C07295=1221.283,24.930,-43.229,-179.294,5.443,148.738
C07296=1221.289,24.681,-43.214,-179.297,5.442,148.739
C07297=1221.293,24.432,-43.199,-179.299,5.442,148.739
C07298=1221.299,24.182,-43.183,-179.302,5.441,148.740
C07299=1221.303,23.932,-43.168,-179.304,5.442,148.741
C07300=1221.308,23.682,-43.153,-179.307,5.441,148.741
C07301=1221.314,23.433,-43.137,-179.309,5.441,148.742
C07302=1221.318,23.184,-43.122,-179.312,5.440,148.743
C07303=1221.324,22.934,-43.107,-179.315,5.439,148.743
C07304=1221.328,22.685,-43.091,-179.317,5.439,148.744
C07305=1221.333,22.435,-43.076,-179.320,5.438,148.745
C07306=1221.338,22.186,-43.061,-179.321,5.438,148.745
C07307=1221.343,21.936,-43.046,-179.324,5.438,148.746
C07308=1221.348,21.687,-43.031,-179.327,5.437,148.747
C07309=1221.354,21.438,-43.015,-179.329,5.437,148.747
C07310=1221.358,21.188,-43.000,-179.332,5.436,148.748
C07311=1221.363,20.938,-42.985,-179.335,5.436,148.749
C07312=1221.368,20.689,-42.970,-179.337,5.436,148.749
C07313=1221.373,20.439,-42.955,-179.339,5.435,148.750
C07314=1221.378,20.190,-42.940,-179.342,5.435,148.751
C07315=1221.384,19.940,-42.925,-179.345,5.434,148.751
C07316=1221.388,19.691,-42.910,-179.347,5.434,148.752
C07317=1221.393,19.441,-42.894,-179.350,5.433,148.753
C07318=1221.398,19.192,-42.879,-179.353,5.433,148.753
C07319=1221.403,18.942,-42.864,-179.354,5.433,148.754
C07320=1221.408,18.693,-42.849,-179.357,5.432,148.755
C07321=1221.413,18.443,-42.833,-179.359,5.432,148.755
C07322=1221.418,18.194,-42.819,-179.362,5.431,148.756
C07323=1221.423,17.945,-42.804,-179.365,5.431,148.757
C07324=1221.428,17.695,-42.788,-179.367,5.430,148.757
C07325=1221.433,17.446,-42.774,-179.370,5.430,148.758
C07326=1221.439,17.196,-42.759,-179.372,5.430,148.759
C07327=1221.443,16.946,-42.743,-179.375,5.429,148.759
C07328=1221.449,16.696,-42.728,-179.377,5.429,148.760
C07329=1221.453,16.447,-42.713,-179.380,5.428,148.761
C07330=1221.458,16.198,-42.698,-179.383,5.428,148.761
C07331=1221.464,15.948,-42.683,-179.385,5.428,148.762
C07332=1221.468,15.699,-42.668,-179.387,5.427,148.763
C07333=1221.473,15.449,-42.654,-179.390,5.426,148.763
C07334=1221.479,15.200,-42.639,-179.392,5.426,148.764
C07335=1221.483,14.951,-42.624,-179.395,5.425,148.765
C07336=1221.489,14.701,-42.609,-179.397,5.426,148.765
C07337=1221.493,14.452,-42.594,-179.400,5.425,148.766
C07338=1221.498,14.202,-42.579,-179.402,5.425,148.767
C07339=1221.504,13.953,-42.564,-179.405,5.424,148.767
C07340=1221.509,13.703,-42.550,-179.408,5.424,148.768
C07341=1221.513,13.454,-42.535,-179.410,5.423,148.769
C07342=1221.519,13.204,-42.519,-179.412,5.423,148.769
C07343=1221.523,12.954,-42.504,-179.415,5.423,148.770
C07344=1221.528,12.705,-42.489,-179.418,5.422,148.771
C07345=1221.534,12.455,-42.474,-179.420,5.422,148.771
C07346=1221.538,12.206,-42.459,-179.423,5.421,148.772
C07347=1221.543,11.956,-42.445,-179.425,5.421,148.773
C07348=1221.548,11.707,-42.430,-179.428,5.421,148.773
C07349=1221.553,11.457,-42.415,-179.430,5.420,148.774
C07350=1221.558,11.207,-42.401,-179.432,5.420,148.775
C07351=1221.563,10.958,-42.386,-179.435,5.419,148.775
C07352=1221.569,10.708,-42.371,-179.437,5.419,148.776
C07353=1221.573,10.459,-42.356,-179.440,5.419,148.777
C07354=1221.578,10.209,-42.342,-179.442,5.418,148.777
C07355=1221.583,9.960,-42.327,-179.445,5.418,148.778
C07356=1221.589,9.710,-42.312,-179.448,5.417,148.779
C07357=1221.593,9.461,-42.297,-179.450,5.417,148.779
C07358=1221.598,9.211,-42.283,-179.452,5.417,148.780
C07359=1221.604,8.962,-42.269,-179.455,5.416,148.781
C07360=1221.609,8.713,-42.253,-179.458,5.416,148.781
C07361=1221.614,8.463,-42.239,-179.460,5.415,148.782
C07362=1221.619,8.214,-42.225,-179.463,5.416,148.783
C07363=1221.624,7.964,-42.210,-179.465,5.415,148.784
C07364=1221.629,7.715,-42.195,-179.468,5.415,148.784
C07365=1221.634,7.465,-42.180,-179.470,5.414,148.785
C07366=1221.639,7.216,-42.166,-179.473,5.414,148.786
C07367=1221.644,6.966,-42.151,-179.475,5.414,148.786
C07368=1221.649,6.717,-42.136,-179.477,5.413,148.787
C07369=1221.654,6.467,-42.122,-179.480,5.412,148.787
C07370=1221.659,6.217,-42.108,-179.483,5.412,148.788
C07371=1221.664,5.967,-42.093,-179.485,5.411,148.789
C07372=1221.669,5.718,-42.078,-179.487,5.412,148.789
C07373=1221.674,5.469,-42.064,-179.490,5.411,148.790
C07374=1221.679,5.219,-42.049,-179.493,5.411,148.791
C07375=1221.684,4.970,-42.034,-179.495,5.410,148.792
C07376=1221.689,4.721,-42.020,-179.497,5.410,148.792
C07377=1221.695,4.471,-42.006,-179.500,5.410,148.793
C07378=1221.700,4.221,-41.991,-179.503,5.409,148.794
C07379=1221.704,3.972,-41.976,-179.505,5.409,148.794
C07380=1221.710,3.703,-41.961,-179.508,5.408,148.795
C07381=1221.715,3.434,-41.946,-179.511,5.408,148.796
C07382=1221.720,3.165,-41.930,-179.514,5.408,148.797
C07383=1221.726,2.895,-41.914,-179.516,5.408,148.797
C07384=1221.731,2.646,-41.899,-179.519,5.407,148.798
C07385=1221.736,2.396,-41.885,-179.521,5.407,148.799
C07386=1221.741,2.147,-41.871,-179.524,5.406,148.799
C07387=1221.746,1.898,-41.857,-179.527,5.406,148.800
C07388=1221.751,1.648,-41.843,-179.529,5.406,148.801
C07389=1221.756,1.399,-41.828,-179.531,5.405,148.801
C07390=1221.761,1.149,-41.813,-179.533,5.405,148.802
C07391=1221.766,0.900,-41.799,-179.536,5.404,148.803
C07392=1221.771,0.650,-41.785,-179.538,5.405,148.803
C07393=1221.776,0.401,-41.771,-179.541,5.404,148.804
C07394=1221.781,0.151,-41.757,-179.543,5.404,148.805
C07395=1221.786,-0.099,-41.742,-179.546,5.403,148.805
C07396=1221.791,-0.348,-41.728,-179.548,5.403,148.806
C07397=1221.796,-0.597,-41.713,-179.551,5.403,148.807
C07398=1221.801,-0.847,-41.699,-179.553,5.402,148.807
C07399=1221.806,-1.096,-41.685,-179.556,5.402,148.808
C07400=1221.811,-1.346,-41.671,-179.558,5.402,148.809
C07401=1221.816,-1.596,-41.656,-179.561,5.402,148.809
C07402=1221.821,-1.845,-41.642,-179.563,5.401,148.810
C07403=1221.826,-2.095,-41.628,-179.566,5.400,148.811
C07404=1221.832,-2.344,-41.614,-179.568,5.401,148.811
C07405=1221.837,-2.594,-41.600,-179.571,5.400,148.812
C07406=1221.842,-2.843,-41.585,-179.574,5.400,148.813
C07407=1221.847,-3.093,-41.571,-179.576,5.399,148.814
C07408=1221.852,-3.343,-41.557,-179.578,5.400,148.814
C07409=1221.857,-3.592,-41.543,-179.581,5.399,148.815
C07410=1221.862,-3.842,-41.529,-179.584,5.399,148.816
C07411=1221.867,-4.091,-41.514,-179.586,5.398,148.816
C07412=1221.872,-4.341,-41.500,-179.588,5.398,148.817
C07413=1221.877,-4.591,-41.486,-179.591,5.398,148.818
C07414=1221.883,-4.840,-41.472,-179.594,5.397,148.818
C07415=1221.887,-5.089,-41.458,-179.596,5.397,148.819
C07416=1221.892,-5.339,-41.443,-179.598,5.397,148.820
C07417=1221.897,-5.589,-41.429,-179.601,5.396,148.820
C07418=1221.902,-5.838,-41.416,-179.603,5.396,148.821
C07419=1221.907,-6.087,-41.401,-179.606,5.395,148.822
C07420=1221.912,-6.337,-41.387,-179.608,5.395,148.822
C07421=1221.917,-6.587,-41.374,-179.611,5.395,148.823
C07422=1221.923,-6.836,-41.360,-179.613,5.394,148.824
C07423=1221.928,-7.086,-41.345,-179.616,5.394,148.824
C07424=1221.933,-7.336,-41.331,-179.618,5.394,148.825
C07425=1221.938,-7.585,-41.317,-179.621,5.394,148.826
C07426=1221.943,-7.834,-41.303,-179.623,5.393,148.826
C07427=1221.948,-8.084,-41.289,-179.626,5.393,148.827
C07428=1221.953,-8.334,-41.275,-179.628,5.393,148.828
C07429=1221.958,-8.583,-41.261,-179.631,5.392,148.829
C07430=1221.963,-8.833,-41.247,-179.633,5.392,148.829
C07431=1221.968,-9.083,-41.233,-179.635,5.392,148.830
C07432=1221.973,-9.332,-41.219,-179.638,5.392,148.831
C07433=1221.978,-9.581,-41.206,-179.641,5.391,148.831
C07434=1221.983,-9.831,-41.191,-179.643,5.391,148.832
C07435=1221.988,-10.081,-41.178,-179.645,5.391,148.833
C07436=1221.994,-10.330,-41.164,-179.648,5.391,148.833
C07437=1221.999,-10.580,-41.150,-179.651,5.390,148.834
C07438=1222.003,-10.829,-41.136,-179.653,5.390,148.835
C07439=1222.008,-11.079,-41.122,-179.655,5.390,148.835
C07440=1222.014,-11.328,-41.108,-179.658,5.389,148.836
C07441=1222.019,-11.578,-41.094,-179.661,5.389,148.837
C07442=1222.023,-11.828,-41.080,-179.663,5.389,148.838
C07443=1222.029,-12.077,-41.067,-179.666,5.389,148.838
C07444=1222.034,-12.327,-41.053,-179.668,5.388,148.839
C07445=1222.039,-12.577,-41.039,-179.671,5.388,148.840
C07446=1222.044,-12.825,-41.025,-179.673,5.388,148.840
C07447=1222.049,-13.076,-41.012,-179.676,5.387,148.841
C07448=1222.054,-13.325,-40.998,-179.678,5.387,148.842
C07449=1222.059,-13.574,-40.984,-179.680,5.387,148.842
C07450=1222.064,-13.824,-40.970,-179.683,5.387,148.843
C07451=1222.069,-14.073,-40.957,-179.686,5.386,148.844
C07452=1222.074,-14.323,-40.942,-179.688,5.386,148.844
C07453=1222.079,-14.573,-40.928,-179.690,5.386,148.845
C07454=1222.084,-14.822,-40.916,-179.693,5.385,148.846
C07455=1222.089,-15.072,-40.901,-179.696,5.385,148.847
C07456=1222.094,-15.322,-40.887,-179.698,5.385,148.847
C07457=1222.099,-15.571,-40.874,-179.700,5.384,148.848
C07458=1222.104,-15.821,-40.860,-179.703,5.384,148.848
C07459=1222.110,-16.070,-40.847,-179.705,5.384,148.849
C07460=1222.115,-16.320,-40.833,-179.707,5.384,148.850
C07461=1222.119,-16.569,-40.819,-179.710,5.383,148.850
C07462=1222.125,-16.819,-40.806,-179.713,5.383,148.851
C07463=1222.130,-17.068,-40.792,-179.715,5.383,148.852
C07464=1222.135,-17.318,-40.779,-179.717,5.383,148.853
C07465=1222.140,-17.568,-40.765,-179.720,5.382,148.853
C07466=1222.145,-17.817,-40.751,-179.722,5.382,148.854
C07467=1222.150,-18.067,-40.738,-179.725,5.382,148.855
C07468=1222.155,-18.316,-40.723,-179.727,5.381,148.855
C07469=1222.161,-18.566,-40.711,-179.729,5.382,148.856
C07470=1222.165,-18.815,-40.697,-179.732,5.381,148.857
C07471=1222.171,-19.065,-40.683,-179.735,5.381,148.857
C07472=1222.176,-19.315,-40.670,-179.737,5.380,148.858
C07473=1222.181,-19.565,-40.656,-179.740,5.380,148.859
C07474=1222.186,-19.814,-40.643,-179.742,5.380,148.860
C07475=1222.191,-20.064,-40.629,-179.745,5.379,148.860
C07476=1222.196,-20.313,-40.615,-179.747,5.380,148.861
C07477=1222.201,-20.563,-40.602,-179.750,5.379,148.862
C07478=1222.207,-20.812,-40.589,-179.752,5.379,148.862
C07479=1222.211,-21.062,-40.576,-179.754,5.379,148.863
C07480=1222.217,-21.311,-40.562,-179.757,5.379,148.864
C07481=1222.221,-21.561,-40.549,-179.760,5.378,148.864
C07482=1222.227,-21.810,-40.535,-179.762,5.378,148.865
C07483=1222.232,-22.060,-40.521,-179.764,5.378,148.866
C07484=1222.237,-22.329,-40.507,-179.767,5.377,148.866
C07485=1222.243,-22.599,-40.493,-179.770,5.377,148.867
C07486=1222.248,-22.868,-40.478,-179.773,5.377,148.868
C07487=1222.253,-23.137,-40.463,-179.775,5.377,148.869
C07488=1222.259,-23.387,-40.450,-179.778,5.377,148.869
C07489=1222.264,-23.637,-40.437,-179.780,5.376,148.870
C07490=1222.269,-23.886,-40.423,-179.782,5.376,148.871
C07491=1222.274,-24.136,-40.410,-179.785,5.376,148.872
C07492=1222.279,-24.386,-40.397,-179.788,5.375,148.872
C07493=1222.284,-24.635,-40.384,-179.790,5.376,148.873
C07494=1222.290,-24.885,-40.370,-179.792,5.375,148.874
C07495=1222.294,-25.134,-40.357,-179.795,5.375,148.874
C07496=1222.300,-25.384,-40.343,-179.797,5.375,148.875
C07497=1222.304,-25.634,-40.331,-179.800,5.375,148.876
C07498=1222.310,-25.883,-40.317,-179.802,5.374,148.876
C07499=1222.314,-26.133,-40.304,-179.805,5.374,148.877
C07500=1222.320,-26.382,-40.290,-179.807,5.374,148.878
C07501=1222.325,-26.632,-40.277,-179.810,5.373,148.879
C07502=1222.330,-26.881,-40.264,-179.812,5.374,148.879
C07503=1222.335,-27.131,-40.251,-179.815,5.373,148.880
C07504=1222.340,-27.381,-40.238,-179.817,5.373,148.881
C07505=1222.345,-27.630,-40.224,-179.819,5.373,148.881
C07506=1222.350,-27.880,-40.211,-179.822,5.372,148.882
C07507=1222.356,-28.129,-40.198,-179.825,5.372,148.883
C07508=1222.360,-28.379,-40.185,-179.827,5.372,148.883
C07509=1222.366,-28.628,-40.171,-179.829,5.372,148.884
C07510=1222.370,-28.878,-40.158,-179.832,5.371,148.885
C07511=1222.375,-29.128,-40.145,-179.834,5.372,148.886
C07512=1222.381,-29.378,-40.132,-179.837,5.371,148.886
C07513=1222.386,-29.627,-40.119,-179.839,5.371,148.887
C07514=1222.391,-29.876,-40.105,-179.842,5.371,148.888
C07515=1222.396,-30.126,-40.092,-179.844,5.370,148.888
C07516=1222.401,-30.376,-40.080,-179.847,5.370,148.889
C07517=1222.406,-30.626,-40.066,-179.849,5.370,148.890
C07518=1222.411,-30.875,-40.054,-179.852,5.370,148.890
C07519=1222.416,-31.124,-40.040,-179.854,5.369,148.891
C07520=1222.422,-31.374,-40.027,-179.856,5.369,148.892
C07521=1222.427,-31.624,-40.014,-179.859,5.369,148.892
C07522=1222.431,-31.874,-40.001,-179.861,5.368,148.893
C07523=1222.437,-32.123,-39.988,-179.863,5.369,148.894
C07524=1222.442,-32.373,-39.975,-179.866,5.368,148.894
C07525=1222.447,-32.623,-39.962,-179.869,5.368,148.895
C07526=1222.453,-32.872,-39.949,-179.871,5.368,148.896
C07527=1222.457,-33.121,-39.936,-179.873,5.367,148.896
C07528=1222.462,-33.371,-39.923,-179.876,5.367,148.897
C07529=1222.468,-33.621,-39.910,-179.878,5.367,148.898
C07530=1222.473,-33.870,-39.897,-179.881,5.367,148.899
C07531=1222.477,-34.120,-39.884,-179.883,5.367,148.899
C07532=1222.483,-34.370,-39.871,-179.885,5.367,148.900
C07533=1222.488,-34.620,-39.858,-179.888,5.366,148.901
C07534=1222.493,-34.869,-39.845,-179.890,5.366,148.901
C07535=1222.498,-35.118,-39.833,-179.893,5.366,148.902
C07536=1222.503,-35.369,-39.819,-179.896,5.365,148.903
C07537=1222.508,-35.618,-39.807,-179.898,5.366,148.903
C07538=1222.514,-35.867,-39.794,-179.900,5.365,148.904
C07539=1222.518,-36.117,-39.781,-179.903,5.365,148.905
C07540=1222.524,-36.367,-39.768,-179.905,5.365,148.906
C07541=1222.529,-36.616,-39.755,-179.908,5.365,148.906
C07542=1222.534,-36.865,-39.743,-179.910,5.365,148.907
C07543=1222.539,-37.116,-39.730,-179.912,5.365,148.908
C07544=1222.545,-37.365,-39.717,-179.915,5.364,148.908
C07545=1222.550,-37.614,-39.704,-179.917,5.364,148.909
C07546=1222.554,-37.864,-39.691,-179.920,5.364,148.910
C07547=1222.559,-38.114,-39.678,-179.923,5.363,148.910
C07548=1222.565,-38.363,-39.665,-179.925,5.364,148.911
C07549=1222.570,-38.613,-39.652,-179.927,5.363,148.912
C07550=1222.575,-38.863,-39.640,-179.930,5.363,148.913
C07551=1222.580,-39.112,-39.627,-179.932,5.363,148.913
C07552=1222.585,-39.361,-39.614,-179.935,5.363,148.914
C07553=1222.590,-39.612,-39.601,-179.937,5.363,148.915
C07554=1222.595,-39.861,-39.588,-179.939,5.362,148.915
C07555=1222.601,-40.110,-39.576,-179.942,5.362,148.916
C07556=1222.605,-40.361,-39.563,-179.944,5.362,148.917
C07557=1222.611,-40.610,-39.551,-179.947,5.362,148.917
C07558=1222.616,-40.860,-39.538,-179.950,5.361,148.918
C07559=1222.621,-41.109,-39.526,-179.952,5.362,148.919
C07560=1222.626,-41.359,-39.512,-179.954,5.361,148.920
C07561=1222.631,-41.609,-39.499,-179.956,5.361,148.920
C07562=1222.636,-41.858,-39.487,-179.959,5.361,148.921
C07563=1222.642,-42.108,-39.475,-179.962,5.360,148.922
C07564=1222.646,-42.358,-39.462,-179.964,5.361,148.922
C07565=1222.651,-42.607,-39.449,-179.966,5.360,148.923
C07566=1222.656,-42.857,-39.437,-179.969,5.360,148.924
C07567=1222.662,-43.106,-39.424,-179.971,5.360,148.924
C07568=1222.667,-43.355,-39.411,-179.974,5.360,148.925
C07569=1222.672,-43.606,-39.399,-179.976,5.360,148.926
C07570=1222.677,-43.855,-39.386,-179.979,5.360,148.927
C07571=1222.683,-44.105,-39.374,-179.981,5.359,148.927
C07572=1222.688,-44.354,-39.361,-179.983,5.359,148.928
C07573=1222.692,-44.605,-39.349,-179.986,5.359,148.929
C07574=1222.698,-44.854,-39.336,-179.988,5.359,148.929
C07575=1222.703,-45.103,-39.324,-179.991,5.359,148.930
C07576=1222.708,-45.353,-39.311,-179.993,5.358,148.931
C07577=1222.713,-45.603,-39.299,-179.995,5.359,148.931
C07578=1222.718,-45.853,-39.286,-179.998,5.358,148.932
C07579=1222.723,-46.102,-39.273,179.999,5.358,148.933
C07580=1222.728,-46.351,-39.261,179.997,5.358,148.934
C07581=1222.733,-46.601,-39.249,179.994,5.357,148.934
C07582=1222.739,-46.850,-39.236,179.992,5.358,148.935
C07583=1222.744,-47.100,-39.224,179.990,5.357,148.936
C07584=1222.749,-47.350,-39.212,179.987,5.357,148.936
C07585=1222.754,-47.600,-39.198,179.985,5.357,148.937
C07586=1222.760,-47.849,-39.186,179.982,5.357,148.938
C07587=1222.765,-48.099,-39.174,179.980,5.357,148.938
C07588=1222.770,-48.369,-39.160,179.978,5.357,148.939
C07589=1222.776,-48.638,-39.147,179.975,5.356,148.940
C07590=1222.781,-48.908,-39.134,179.972,5.356,148.941
C07591=1222.787,-49.178,-39.120,179.970,5.356,148.942
C07592=1222.792,-49.428,-39.108,179.967,5.356,148.942
C07593=1222.797,-49.678,-39.095,179.965,5.356,148.943
C07594=1222.803,-49.928,-39.083,179.963,5.355,148.943
C07595=1222.807,-50.177,-39.071,179.960,5.355,148.944
C07596=1222.812,-50.426,-39.059,179.958,5.355,148.945
C07597=1222.817,-50.677,-39.046,179.955,5.355,148.946
C07598=1222.822,-50.926,-39.034,179.953,5.355,148.946
C07599=1222.828,-51.176,-39.022,179.951,5.355,148.947
C07600=1222.833,-51.425,-39.009,179.948,5.354,148.948
C07601=1222.838,-51.675,-38.997,179.946,5.354,148.948
C07602=1222.843,-51.924,-38.985,179.943,5.354,148.949
C07603=1222.848,-52.174,-38.972,179.941,5.354,148.950
C07604=1222.854,-52.424,-38.960,179.938,5.354,148.950
C07605=1222.859,-52.673,-38.948,179.936,5.353,148.951
C07606=1222.864,-52.924,-38.935,179.934,5.354,148.952
C07607=1222.869,-53.173,-38.923,179.931,5.353,148.953
C07608=1222.874,-53.423,-38.912,179.929,5.354,148.953
C07609=1222.879,-53.672,-38.899,179.926,5.353,148.954
C07610=1222.884,-53.922,-38.887,179.923,5.353,148.955
C07611=1222.889,-54.171,-38.874,179.921,5.353,148.955
C07612=1222.895,-54.421,-38.863,179.919,5.352,148.956
C07613=1222.900,-54.670,-38.850,179.917,5.353,148.957
C07614=1222.905,-54.920,-38.838,179.914,5.352,148.957
C07615=1222.910,-55.169,-38.826,179.912,5.353,148.958
C07616=1222.915,-55.419,-38.814,179.909,5.352,148.959
C07617=1222.920,-55.669,-38.802,179.907,5.352,148.960
C07618=1222.926,-55.919,-38.790,179.904,5.352,148.960
C07619=1222.930,-56.169,-38.777,179.902,5.352,148.961
C07620=1222.935,-56.419,-38.765,179.900,5.352,148.962
C07621=1222.940,-56.668,-38.754,179.897,5.351,148.962
C07622=1222.945,-56.917,-38.741,179.894,5.351,148.963
C07623=1222.951,-57.167,-38.729,179.892,5.351,148.964
C07624=1222.956,-57.417,-38.717,179.890,5.351,148.965
C07625=1222.961,-57.667,-38.705,179.888,5.351,148.965
C07626=1222.966,-57.916,-38.693,179.885,5.351,148.966
C07627=1222.971,-58.166,-38.681,179.883,5.351,148.967
C07628=1222.977,-58.416,-38.669,179.880,5.351,148.967
C07629=1222.982,-58.665,-38.657,179.877,5.350,148.968
C07630=1222.987,-58.915,-38.644,179.875,5.350,148.969
C07631=1222.992,-59.164,-38.633,179.873,5.350,148.969
C07632=1222.997,-59.414,-38.621,179.871,5.350,148.970
C07633=1223.002,-59.664,-38.609,179.868,5.350,148.971
C07634=1223.008,-59.914,-38.597,179.866,5.350,148.972
C07635=1223.012,-60.163,-38.585,179.863,5.350,148.972
C07636=1223.018,-60.413,-38.573,179.861,5.349,148.973
C07637=1223.023,-60.662,-38.561,179.858,5.350,148.974
C07638=1223.028,-60.912,-38.549,179.856,5.349,148.974
C07639=1223.033,-61.161,-38.537,179.854,5.349,148.975
C07640=1223.038,-61.411,-38.525,179.851,5.349,148.976
C07641=1223.044,-61.661,-38.513,179.849,5.349,148.976
C07642=1223.048,-61.911,-38.502,179.847,5.349,148.977
C07643=1223.053,-62.160,-38.489,179.844,5.348,148.978
C07644=1223.059,-62.410,-38.477,179.842,5.348,148.978
C07645=1223.064,-62.660,-38.466,179.839,5.348,148.979
C07646=1223.069,-62.910,-38.454,179.837,5.348,148.980
C07647=1223.074,-63.159,-38.442,179.835,5.348,148.981
C07648=1223.080,-63.409,-38.430,179.833,5.348,148.981
C07649=1223.084,-63.659,-38.419,179.830,5.348,148.982
C07650=1223.090,-63.908,-38.407,179.828,5.348,148.983
C07651=1223.095,-64.157,-38.394,179.825,5.348,148.983
C07652=1223.100,-64.407,-38.383,179.822,5.347,148.984
C07653=1223.106,-64.657,-38.371,179.820,5.347,148.985
C07654=1223.111,-64.907,-38.359,179.818,5.347,148.985
C07655=1223.116,-65.156,-38.348,179.816,5.347,148.986
C07656=1223.121,-65.406,-38.336,179.813,5.347,148.987
C07657=1223.126,-65.656,-38.324,179.811,5.347,148.988
C07658=1223.131,-65.905,-38.312,179.808,5.347,148.988
C07659=1223.136,-66.155,-38.300,179.806,5.347,148.989
C07660=1223.141,-66.405,-38.289,179.803,5.347,148.990
C07661=1223.146,-66.655,-38.277,179.801,5.346,148.990
C07662=1223.152,-66.905,-38.265,179.799,5.347,148.991
C07663=1223.157,-67.154,-38.254,179.796,5.346,148.992
C07664=1223.162,-67.403,-38.242,179.794,5.346,148.993
C07665=1223.167,-67.652,-38.231,179.791,5.346,148.993
C07666=1223.172,-67.902,-38.219,179.789,5.346,148.994
C07667=1223.178,-68.152,-38.207,179.786,5.346,148.995
C07668=1223.183,-68.402,-38.195,179.784,5.346,148.995
C07669=1223.188,-68.652,-38.184,179.782,5.346,148.996
C07670=1223.193,-68.902,-38.172,179.779,5.345,148.997
C07671=1223.198,-69.151,-38.160,179.777,5.346,148.997
C07672=1223.204,-69.401,-38.149,179.775,5.345,148.998
C07673=1223.209,-69.650,-38.138,179.773,5.345,148.999
C07674=1223.214,-69.900,-38.126,179.770,5.345,148.999
C07675=1223.219,-70.150,-38.114,179.768,5.345,149.000
C07676=1223.224,-70.400,-38.103,179.765,5.345,149.001
C07677=1223.229,-70.649,-38.091,179.763,5.345,149.001
C07678=1223.235,-70.899,-38.079,179.760,5.344,149.002
C07679=1223.240,-71.148,-38.068,179.758,5.345,149.003
C07680=1223.245,-71.398,-38.057,179.756,5.344,149.004
C07681=1223.250,-71.648,-38.045,179.753,5.344,149.004
C07682=1223.255,-71.898,-38.033,179.751,5.344,149.005
C07683=1223.260,-72.147,-38.022,179.748,5.344,149.006
C07684=1223.265,-72.397,-38.010,179.746,5.344,149.006
C07685=1223.271,-72.646,-37.999,179.744,5.344,149.007
C07686=1223.276,-72.896,-37.987,179.741,5.344,149.008
C07687=1223.281,-73.146,-37.976,179.739,5.344,149.009
C07688=1223.286,-73.396,-37.964,179.737,5.344,149.009
C07689=1223.291,-73.645,-37.953,179.734,5.343,149.010
C07690=1223.297,-73.895,-37.941,179.732,5.344,149.011
C07691=1223.302,-74.144,-37.930,179.729,5.343,149.011
C07692=1223.307,-74.415,-37.918,179.727,5.343,149.012
C07693=1223.313,-74.685,-37.905,179.724,5.343,149.013
C07694=1223.319,-74.956,-37.893,179.722,5.343,149.014
C07695=1223.324,-75.226,-37.880,179.719,5.342,149.014
C07696=1223.330,-75.476,-37.870,179.717,5.343,149.015
C07697=1223.335,-75.726,-37.858,179.714,5.342,149.016
C07698=1223.340,-75.975,-37.847,179.712,5.343,149.016
C07699=1223.345,-76.225,-37.835,179.710,5.342,149.017
C07700=1223.350,-76.475,-37.823,179.708,5.342,149.018
C07701=1223.356,-76.724,-37.812,179.705,5.342,149.018
C07702=1223.361,-76.974,-37.801,179.703,5.342,149.019
C07703=1223.366,-77.224,-37.790,179.700,5.342,149.020
C07704=1223.371,-77.474,-37.778,179.698,5.342,149.021
C07705=1223.376,-77.723,-37.767,179.695,5.342,149.021
C07706=1223.382,-77.973,-37.755,179.693,5.342,149.022
C07707=1223.387,-78.222,-37.744,179.691,5.342,149.023
C07708=1223.392,-78.473,-37.734,179.688,5.342,149.023
C07709=1223.398,-78.722,-37.722,179.686,5.342,149.024
C07710=1223.402,-78.972,-37.711,179.683,5.341,149.025
C07711=1223.408,-79.221,-37.699,179.681,5.341,149.026
C07712=1223.412,-79.471,-37.688,179.678,5.341,149.026
C07713=1223.418,-79.721,-37.677,179.676,5.341,149.027
C07714=1223.423,-79.971,-37.665,179.674,5.341,149.027
C07715=1223.428,-80.220,-37.654,179.672,5.341,149.028
C07716=1223.433,-80.469,-37.643,179.669,5.340,149.029
C07717=1223.439,-80.720,-37.632,179.667,5.341,149.030
C07718=1223.444,-80.969,-37.621,179.665,5.340,149.030
C07719=1223.449,-81.219,-37.610,179.663,5.341,149.031
C07720=1223.455,-81.468,-37.598,179.660,5.340,149.032
C07721=1223.460,-81.718,-37.587,179.658,5.341,149.032
C07722=1223.464,-81.968,-37.576,179.655,5.340,149.033
C07723=1223.470,-82.217,-37.565,179.653,5.341,149.034
C07724=1223.475,-82.468,-37.554,179.650,5.340,149.035
C07725=1223.480,-82.717,-37.543,179.648,5.340,149.035
C07726=1223.485,-82.967,-37.531,179.646,5.340,149.036
C07727=1223.491,-83.217,-37.521,179.643,5.340,149.037
C07728=1223.496,-83.466,-37.509,179.641,5.340,149.037
C07729=1223.500,-83.716,-37.498,179.639,5.340,149.038
C07730=1223.506,-83.965,-37.488,179.636,5.340,149.039
C07731=1223.511,-84.215,-37.476,179.634,5.340,149.039
C07732=1223.516,-84.465,-37.465,179.632,5.339,149.040
C07733=1223.522,-84.715,-37.454,179.630,5.340,149.041
C07734=1223.526,-84.964,-37.443,179.627,5.339,149.041
C07735=1223.532,-85.215,-37.432,179.624,5.339,149.042
C07736=1223.537,-85.464,-37.421,179.622,5.339,149.043
C07737=1223.542,-85.713,-37.410,179.620,5.339,149.044
C07738=1223.547,-85.964,-37.399,179.617,5.339,149.044
C07739=1223.553,-86.213,-37.388,179.615,5.339,149.045
C07740=1223.558,-86.463,-37.377,179.613,5.339,149.046
C07741=1223.563,-86.713,-37.366,179.610,5.339,149.046
C07742=1223.568,-86.962,-37.355,179.608,5.339,149.047
C07743=1223.573,-87.212,-37.344,179.605,5.338,149.048
C07744=1223.579,-87.461,-37.333,179.603,5.339,149.049
C07745=1223.584,-87.711,-37.322,179.601,5.338,149.049
C07746=1223.589,-87.961,-37.311,179.599,5.338,149.050
C07747=1223.594,-88.210,-37.301,179.596,5.338,149.050
C07748=1223.599,-88.460,-37.289,179.594,5.338,149.051
C07749=1223.605,-88.711,-37.278,179.591,5.338,149.052
C07750=1223.610,-88.960,-37.267,179.589,5.338,149.053
C07751=1223.615,-89.210,-37.257,179.587,5.338,149.053
C07752=1223.620,-89.459,-37.246,179.585,5.338,149.054
C07753=1223.625,-89.709,-37.235,179.582,5.338,149.055
C07754=1223.630,-89.959,-37.224,179.580,5.338,149.055
C07755=1223.637,-90.208,-37.213,179.577,5.338,149.056
C07756=1223.641,-90.458,-37.202,179.575,5.338,149.057
C07757=1223.647,-90.708,-37.192,179.572,5.337,149.058
C07758=1223.651,-90.957,-37.180,179.571,5.337,149.058
C07759=1223.657,-91.207,-37.170,179.568,5.337,149.059
C07760=1223.662,-91.456,-37.159,179.566,5.337,149.059
C07761=1223.667,-91.707,-37.148,179.563,5.337,149.060
C07762=1223.672,-91.956,-37.138,179.561,5.337,149.061
C07763=1223.678,-92.206,-37.126,179.559,5.337,149.062
C07764=1223.683,-92.456,-37.116,179.557,5.337,149.062
C07765=1223.688,-92.705,-37.105,179.554,5.337,149.063
C07766=1223.694,-92.955,-37.095,179.552,5.337,149.064
C07767=1223.699,-93.205,-37.084,179.549,5.337,149.064
C07768=1223.704,-93.454,-37.073,179.547,5.337,149.065
C07769=1223.709,-93.704,-37.062,179.544,5.337,149.066
C07770=1223.714,-93.954,-37.051,179.543,5.337,149.066
C07771=1223.719,-94.203,-37.041,179.540,5.336,149.067
C07772=1223.724,-94.454,-37.030,179.538,5.337,149.068
C07773=1223.730,-94.703,-37.019,179.535,5.336,149.068
C07774=1223.735,-94.953,-37.009,179.533,5.336,149.069
C07775=1223.740,-95.202,-36.999,179.531,5.336,149.070
C07776=1223.745,-95.452,-36.987,179.528,5.336,149.071
C07777=1223.751,-95.702,-36.977,179.526,5.336,149.071
C07778=1223.756,-95.952,-36.966,179.524,5.336,149.072
C07779=1223.761,-96.201,-36.955,179.521,5.336,149.073
C07780=1223.766,-96.451,-36.945,179.519,5.336,149.073
C07781=1223.772,-96.701,-36.934,179.517,5.335,149.074
C07782=1223.777,-96.950,-36.923,179.515,5.336,149.075
C07783=1223.782,-97.200,-36.913,179.512,5.335,149.075
C07784=1223.787,-97.450,-36.902,179.510,5.336,149.076
C07785=1223.793,-97.700,-36.892,179.507,5.335,149.077
C07786=1223.798,-97.949,-36.881,179.505,5.336,149.078
C07787=1223.803,-98.199,-36.871,179.503,5.336,149.078
C07788=1223.808,-98.449,-36.860,179.500,5.336,149.079
C07789=1223.814,-98.699,-36.850,179.498,5.336,149.080
C07790=1223.819,-98.948,-36.838,179.496,5.335,149.080
C07791=1223.824,-99.198,-36.828,179.494,5.335,149.081
C07792=1223.829,-99.448,-36.818,179.491,5.335,149.082
C07793=1223.835,-99.698,-36.807,179.489,5.335,149.082
C07794=1223.839,-99.948,-36.797,179.486,5.335,149.083
C07795=1223.844,-100.197,-36.787,179.484,5.335,149.084
C07796=1223.850,-100.468,-36.775,179.482,5.335,149.084
C07797=1223.856,-100.739,-36.764,179.479,5.334,149.085
C07798=1223.862,-101.010,-36.752,179.477,5.335,149.086
C07799=1223.868,-101.281,-36.741,179.474,5.335,149.087
C07800=1223.872,-101.531,-36.731,179.472,5.335,149.087
C07801=1223.877,-101.781,-36.720,179.470,5.334,149.088
C07802=1223.883,-102.030,-36.710,179.467,5.335,149.089
C07803=1223.888,-102.280,-36.699,179.465,5.334,149.089
C07804=1223.893,-102.530,-36.689,179.463,5.335,149.090
C07805=1223.899,-102.779,-36.679,179.460,5.334,149.091
C07806=1223.904,-103.029,-36.668,179.458,5.335,149.092
C07807=1223.909,-103.279,-36.658,179.455,5.334,149.092
C07808=1223.914,-103.529,-36.647,179.453,5.335,149.093
C07809=1223.919,-103.778,-36.638,179.451,5.334,149.093
C07810=1223.924,-104.029,-36.627,179.449,5.334,149.094
C07811=1223.930,-104.278,-36.617,179.446,5.334,149.095
C07812=1223.935,-104.527,-36.606,179.444,5.334,149.096
C07813=1223.940,-104.777,-36.595,179.441,5.334,149.096
C07814=1223.946,-105.027,-36.585,179.439,5.334,149.097
C07815=1223.951,-105.277,-36.575,179.437,5.334,149.098
C07816=1223.956,-105.526,-36.565,179.435,5.334,149.098
C07817=1223.961,-105.776,-36.555,179.433,5.334,149.099
C07818=1223.966,-106.026,-36.544,179.430,5.333,149.100
C07819=1223.972,-106.276,-36.534,179.428,5.334,149.100
C07820=1223.977,-106.525,-36.524,179.425,5.333,149.101
C07821=1223.982,-106.775,-36.513,179.423,5.334,149.102
C07822=1223.987,-107.025,-36.504,179.421,5.333,149.103
C07823=1223.992,-107.275,-36.493,179.419,5.334,149.103
C07824=1223.998,-107.524,-36.483,179.416,5.333,149.104
C07825=1224.004,-107.774,-36.473,179.414,5.333,149.104
C07826=1224.009,-108.024,-36.462,179.412,5.333,149.105
C07827=1224.013,-108.273,-36.452,179.410,5.333,149.106
C07828=1224.019,-108.523,-36.442,179.407,5.333,149.107
C07829=1224.024,-108.773,-36.432,179.405,5.333,149.107
C07830=1224.030,-109.023,-36.421,179.402,5.333,149.108
C07831=1224.035,-109.272,-36.411,179.400,5.333,149.109
C07832=1224.039,-109.522,-36.401,179.397,5.333,149.109
C07833=1224.045,-109.772,-36.391,179.396,5.333,149.110
C07834=1224.051,-110.021,-36.381,179.394,5.333,149.111
C07835=1224.056,-110.272,-36.370,179.391,5.333,149.111
C07836=1224.060,-110.521,-36.361,179.389,5.333,149.112
C07837=1224.066,-110.771,-36.351,179.386,5.333,149.113
C07838=1224.071,-111.021,-36.340,179.384,5.333,149.113
C07839=1224.077,-111.271,-36.330,179.381,5.332,149.114
C07840=1224.082,-111.520,-36.321,179.380,5.332,149.115
C07841=1224.087,-111.770,-36.310,179.377,5.332,149.115
C07842=1224.092,-112.020,-36.300,179.375,5.332,149.116
C07843=1224.097,-112.269,-36.290,179.372,5.332,149.117
C07844=1224.103,-112.519,-36.280,179.370,5.332,149.118
C07845=1224.108,-112.769,-36.269,179.368,5.332,149.118
C07846=1224.114,-113.019,-36.260,179.366,5.332,149.119
C07847=1224.119,-113.268,-36.250,179.363,5.332,149.119
C07848=1224.124,-113.518,-36.240,179.361,5.332,149.120
C07849=1224.129,-113.768,-36.230,179.359,5.332,149.121
C07850=1224.134,-114.017,-36.220,179.356,5.332,149.122
C07851=1224.140,-114.267,-36.210,179.354,5.332,149.122
C07852=1224.145,-114.518,-36.200,179.352,5.332,149.123
C07853=1224.150,-114.767,-36.190,179.350,5.332,149.124
C07854=1224.155,-115.016,-36.180,179.347,5.331,149.124
C07855=1224.160,-115.267,-36.170,179.345,5.332,149.125
C07856=1224.165,-115.516,-36.160,179.343,5.331,149.126
C07857=1224.171,-115.766,-36.150,179.341,5.332,149.126
C07858=1224.177,-116.016,-36.140,179.338,5.331,149.127
C07859=1224.181,-116.266,-36.130,179.336,5.332,149.128
C07860=1224.187,-116.515,-36.120,179.334,5.331,149.128
C07861=1224.193,-116.765,-36.111,179.332,5.331,149.129
C07862=1224.197,-117.014,-36.101,179.329,5.332,149.130
C07863=1224.203,-117.264,-36.091,179.327,5.331,149.130
C07864=1224.207,-117.514,-36.081,179.325,5.332,149.131
C07865=1224.213,-117.764,-36.071,179.322,5.331,149.132
C07866=1224.219,-118.014,-36.061,179.320,5.331,149.132
C07867=1224.224,-118.263,-36.051,179.318,5.331,149.133
C07868=1224.229,-118.513,-36.041,179.316,5.331,149.134
C07869=1224.234,-118.763,-36.032,179.313,5.331,149.135
C07870=1224.239,-119.013,-36.022,179.311,5.331,149.135
C07871=1224.245,-119.262,-36.012,179.308,5.331,149.136
C07872=1224.250,-119.512,-36.003,179.307,5.331,149.136
C07873=1224.255,-119.762,-35.992,179.304,5.331,149.137
C07874=1224.260,-120.011,-35.982,179.302,5.331,149.138
C07875=1224.266,-120.262,-35.973,179.300,5.331,149.139
C07876=1224.271,-120.511,-35.963,179.297,5.331,149.139
C07877=1224.276,-120.760,-35.953,179.295,5.331,149.140
C07878=1224.281,-121.011,-35.944,179.293,5.330,149.141
C07879=1224.287,-121.260,-35.934,179.291,5.330,149.141
C07880=1224.292,-121.510,-35.923,179.288,5.330,149.142
C07881=1224.297,-121.760,-35.915,179.286,5.330,149.143
C07882=1224.303,-122.009,-35.904,179.283,5.330,149.143
C07883=1224.307,-122.259,-35.894,179.282,5.330,149.144
C07884=1224.313,-122.509,-35.885,179.279,5.330,149.145
C07885=1224.318,-122.759,-35.875,179.277,5.330,149.145
C07886=1224.324,-123.009,-35.866,179.275,5.330,149.146
C07887=1224.329,-123.258,-35.856,179.272,5.330,149.147
C07888=1224.335,-123.508,-35.847,179.270,5.330,149.147
C07889=1224.339,-123.758,-35.837,179.268,5.330,149.148
C07890=1224.345,-124.008,-35.826,179.266,5.330,149.149
C07891=1224.350,-124.258,-35.818,179.263,5.330,149.149
C07892=1224.355,-124.507,-35.807,179.261,5.330,149.150
C07893=1224.360,-124.757,-35.798,179.259,5.330,149.151
C07894=1224.366,-125.007,-35.788,179.257,5.329,149.151
C07895=1224.371,-125.256,-35.779,179.255,5.330,149.152
C07896=1224.376,-125.507,-35.769,179.252,5.329,149.153
C07897=1224.381,-125.756,-35.760,179.250,5.330,149.153
C07898=1224.386,-126.006,-35.750,179.247,5.329,149.154
C07899=1224.392,-126.256,-35.741,179.245,5.329,149.155
C07900=1223.970,-126.267,-35.777,179.241,5.333,149.157
C07901=1223.965,-126.017,-35.786,179.243,5.333,149.156
C07902=1223.960,-125.767,-35.796,179.246,5.333,149.155
C07903=1223.955,-125.517,-35.805,179.248,5.333,149.155
C07904=1223.949,-125.267,-35.816,179.250,5.333,149.154
C07905=1223.944,-125.017,-35.825,179.252,5.333,149.153
C07906=1223.939,-124.768,-35.835,179.254,5.333,149.153
C07907=1223.934,-124.518,-35.844,179.257,5.333,149.152
C07908=1223.928,-124.268,-35.854,179.259,5.333,149.151
C07909=1223.923,-124.018,-35.863,179.261,5.333,149.151
C07910=1223.917,-123.769,-35.873,179.263,5.333,149.150
C07911=1223.913,-123.518,-35.882,179.266,5.334,149.149
C07912=1223.907,-123.269,-35.892,179.268,5.333,149.149
C07913=1223.902,-123.020,-35.902,179.271,5.334,149.148
C07914=1223.896,-122.769,-35.912,179.272,5.334,149.147
C07915=1223.891,-122.520,-35.921,179.275,5.334,149.147
C07916=1223.885,-122.270,-35.931,179.277,5.334,149.146
C07917=1223.881,-122.020,-35.941,179.279,5.333,149.145
C07918=1223.876,-121.771,-35.951,179.282,5.334,149.145
C07919=1223.870,-121.521,-35.960,179.283,5.334,149.144
C07920=1223.865,-121.271,-35.970,179.286,5.334,149.143
C07921=1223.860,-121.021,-35.979,179.288,5.334,149.143
C07922=1223.854,-120.772,-35.989,179.291,5.334,149.142
C07923=1223.850,-120.522,-35.999,179.293,5.334,149.141
C07924=1223.844,-120.272,-36.009,179.296,5.334,149.140
C07925=1223.839,-120.022,-36.018,179.297,5.334,149.140
C07926=1223.833,-119.773,-36.028,179.300,5.335,149.139
C07927=1223.828,-119.523,-36.038,179.302,5.334,149.139
C07928=1223.823,-119.273,-36.048,179.304,5.334,149.138
C07929=1223.818,-119.023,-36.058,179.307,5.334,149.137
C07930=1223.813,-118.773,-36.067,179.308,5.334,149.137
C07931=1223.807,-118.524,-36.077,179.311,5.335,149.136
C07932=1223.803,-118.274,-36.087,179.313,5.334,149.135
C07933=1223.797,-118.024,-36.097,179.316,5.335,149.134
C07934=1223.791,-117.774,-36.107,179.318,5.334,149.134
C07935=1223.786,-117.525,-36.116,179.321,5.335,149.133
C07936=1223.781,-117.275,-36.127,179.322,5.335,149.133
C07937=1223.776,-117.025,-36.136,179.325,5.335,149.132
C07938=1223.771,-116.775,-36.146,179.327,5.335,149.131
C07939=1223.765,-116.526,-36.156,179.329,5.334,149.130
C07940=1223.760,-116.277,-36.166,179.332,5.335,149.130
C07941=1223.755,-116.026,-36.176,179.334,5.334,149.129
C07942=1223.749,-115.776,-36.186,179.336,5.335,149.129
C07943=1223.744,-115.527,-36.196,179.338,5.335,149.128
C07944=1223.739,-115.277,-36.206,179.341,5.335,149.127
C07945=1223.734,-115.027,-36.216,179.343,5.335,149.126
C07946=1223.729,-114.777,-36.225,179.346,5.335,149.126
C07947=1223.723,-114.528,-36.236,179.348,5.335,149.125
C07948=1223.717,-114.278,-36.246,179.350,5.335,149.124
C07949=1223.713,-114.028,-36.256,179.352,5.335,149.124
C07950=1223.708,-113.779,-36.266,179.355,5.336,149.123
C07951=1223.702,-113.529,-36.275,179.357,5.335,149.122
C07952=1223.697,-113.279,-36.285,179.359,5.335,149.122
C07953=1223.692,-113.029,-36.296,179.362,5.335,149.121
C07954=1223.686,-112.780,-36.306,179.364,5.335,149.120
C07955=1223.681,-112.530,-36.315,179.366,5.336,149.120
C07956=1223.676,-112.280,-36.326,179.368,5.336,149.119
C07957=1223.671,-112.031,-36.336,179.371,5.336,149.118
C07958=1223.665,-111.780,-36.346,179.373,5.336,149.118
C07959=1223.661,-111.530,-36.356,179.375,5.336,149.117
C07960=1223.655,-111.281,-36.366,179.377,5.336,149.116
C07961=1223.649,-111.031,-36.376,179.380,5.336,149.115
C07962=1223.644,-110.782,-36.386,179.382,5.336,149.115
C07963=1223.639,-110.532,-36.396,179.384,5.336,149.114
C07964=1223.634,-110.282,-36.407,179.387,5.336,149.113
C07965=1223.628,-110.033,-36.417,179.389,5.337,149.113
C07966=1223.624,-109.783,-36.427,179.391,5.336,149.112
C07967=1223.618,-109.533,-36.437,179.393,5.336,149.111
C07968=1223.613,-109.284,-36.447,179.396,5.336,149.111
C07969=1223.608,-109.034,-36.458,179.398,5.336,149.110
C07970=1223.602,-108.784,-36.468,179.400,5.337,149.109
C07971=1223.597,-108.534,-36.477,179.402,5.336,149.109
C07972=1223.592,-108.284,-36.487,179.405,5.337,149.108
C07973=1223.586,-108.034,-36.498,179.407,5.336,149.107
C07974=1223.581,-107.784,-36.508,179.410,5.337,149.107
C07975=1223.577,-107.535,-36.518,179.412,5.336,149.106
C07976=1223.571,-107.285,-36.528,179.414,5.337,149.105
C07977=1223.566,-107.035,-36.539,179.416,5.337,149.105
C07978=1223.560,-106.786,-36.549,179.419,5.337,149.104
C07979=1223.555,-106.536,-36.559,179.421,5.337,149.103
C07980=1223.550,-106.286,-36.570,179.424,5.337,149.102
C07981=1223.545,-106.037,-36.579,179.426,5.337,149.102
C07982=1223.540,-105.788,-36.590,179.428,5.337,149.101
C07983=1223.535,-105.537,-36.601,179.431,5.337,149.100
C07984=1223.529,-105.288,-36.611,179.433,5.338,149.100
C07985=1223.524,-105.038,-36.621,179.435,5.337,149.099
C07986=1223.518,-104.788,-36.632,179.437,5.337,149.098
C07987=1223.514,-104.539,-36.641,179.440,5.338,149.098
C07988=1223.509,-104.289,-36.652,179.442,5.337,149.097
C07989=1223.503,-104.039,-36.662,179.444,5.338,149.096
C07990=1223.498,-103.789,-36.673,179.446,5.337,149.096
C07991=1223.492,-103.539,-36.683,179.449,5.338,149.095
C07992=1223.487,-103.290,-36.693,179.451,5.338,149.094
C07993=1223.482,-103.039,-36.704,179.453,5.338,149.094
C07994=1223.477,-102.791,-36.714,179.456,5.338,149.093
C07995=1223.472,-102.541,-36.725,179.458,5.338,149.092
C07996=1223.467,-102.291,-36.735,179.460,5.338,149.092
C07997=1223.462,-102.041,-36.745,179.463,5.338,149.091
C07998=1223.456,-101.791,-36.756,179.465,5.338,149.090
C07999=1223.450,-101.542,-36.766,179.468,5.338,149.089
C08000=1223.445,-101.291,-36.776,179.470,5.338,149.089
C08001=1223.441,-101.021,-36.788,179.473,5.338,149.088
C08002=1223.434,-100.750,-36.799,179.475,5.338,149.087
C08003=1223.429,-100.479,-36.810,179.477,5.338,149.087
C08004=1223.423,-100.208,-36.822,179.480,5.339,149.086
C08005=1223.418,-99.958,-36.833,179.482,5.338,149.085
C08006=1223.413,-99.708,-36.843,179.485,5.339,149.084
C08007=1223.407,-99.458,-36.853,179.487,5.339,149.084
C08008=1223.402,-99.208,-36.864,179.489,5.339,149.083
C08009=1223.397,-98.959,-36.875,179.492,5.339,149.082
C08010=1223.392,-98.709,-36.885,179.494,5.339,149.082
C08011=1223.386,-98.459,-36.896,179.496,5.339,149.081
C08012=1223.381,-98.210,-36.906,179.499,5.339,149.080
C08013=1223.376,-97.960,-36.917,179.501,5.339,149.080
C08014=1223.370,-97.711,-36.927,179.503,5.339,149.079
C08015=1223.365,-97.460,-36.938,179.505,5.339,149.078
C08016=1223.360,-97.211,-36.948,179.507,5.339,149.077
C08017=1223.355,-96.961,-36.959,179.510,5.339,149.077
C08018=1223.349,-96.712,-36.970,179.512,5.339,149.076
C08019=1223.344,-96.461,-36.980,179.515,5.339,149.075
C08020=1223.339,-96.212,-36.991,179.517,5.339,149.075
C08021=1223.334,-95.962,-37.002,179.519,5.340,149.074
C08022=1223.329,-95.713,-37.012,179.521,5.339,149.073
C08023=1223.324,-95.462,-37.022,179.524,5.340,149.073
C08024=1223.318,-95.214,-37.033,179.526,5.339,149.072
C08025=1223.313,-94.963,-37.044,179.529,5.340,149.071
C08026=1223.308,-94.714,-37.054,179.531,5.340,149.071
C08027=1223.303,-94.464,-37.065,179.533,5.340,149.070
C08028=1223.298,-94.214,-37.076,179.536,5.340,149.069
C08029=1223.292,-93.964,-37.086,179.538,5.340,149.068
C08030=1223.288,-93.715,-37.098,179.540,5.340,149.068
C08031=1223.282,-93.465,-37.108,179.543,5.341,149.067
C08032=1223.277,-93.216,-37.119,179.545,5.340,149.067
C08033=1223.272,-92.966,-37.129,179.547,5.341,149.066
C08034=1223.266,-92.715,-37.140,179.549,5.340,149.065
C08035=1223.261,-92.467,-37.151,179.552,5.341,149.064
C08036=1223.256,-92.216,-37.162,179.554,5.340,149.064
C08037=1223.250,-91.967,-37.173,179.557,5.341,149.063
C08038=1223.245,-91.717,-37.183,179.559,5.340,149.062
C08039=1223.240,-91.467,-37.194,179.562,5.341,149.062
C08040=1223.235,-91.218,-37.205,179.564,5.340,149.061
C08041=1223.230,-90.968,-37.215,179.566,5.341,149.060
C08042=1223.225,-90.719,-37.226,179.568,5.341,149.060
C08043=1223.219,-90.468,-37.238,179.571,5.341,149.059
C08044=1223.214,-90.219,-37.248,179.573,5.341,149.058
C08045=1223.209,-89.969,-37.259,179.575,5.341,149.058
C08046=1223.204,-89.719,-37.270,179.577,5.341,149.057
C08047=1223.199,-89.470,-37.281,179.580,5.342,149.056
C08048=1223.194,-89.220,-37.292,179.582,5.341,149.055
C08049=1223.188,-88.971,-37.302,179.585,5.342,149.055
C08050=1223.183,-88.721,-37.314,179.587,5.341,149.054
C08051=1223.178,-88.470,-37.325,179.590,5.342,149.053
C08052=1223.173,-88.222,-37.335,179.592,5.341,149.053
C08053=1223.168,-87.971,-37.346,179.594,5.342,149.052
C08054=1223.163,-87.722,-37.357,179.596,5.342,149.051
C08055=1223.157,-87.472,-37.368,179.599,5.342,149.051
C08056=1223.152,-87.222,-37.379,179.601,5.342,149.050
C08057=1223.146,-86.973,-37.390,179.603,5.342,149.049
C08058=1223.142,-86.723,-37.401,179.606,5.342,149.049
C08059=1223.137,-86.473,-37.411,179.608,5.342,149.048
C08060=1223.131,-86.224,-37.422,179.610,5.342,149.047
C08061=1223.126,-85.974,-37.434,179.613,5.343,149.046
C08062=1223.121,-85.724,-37.445,179.616,5.343,149.046
C08063=1223.116,-85.475,-37.456,179.618,5.343,149.045
C08064=1223.111,-85.225,-37.466,179.620,5.343,149.044
C08065=1223.105,-84.975,-37.478,179.623,5.343,149.044
C08066=1223.100,-84.726,-37.489,179.625,5.343,149.043
C08067=1223.095,-84.475,-37.500,179.627,5.343,149.042
C08068=1223.090,-84.226,-37.511,179.629,5.344,149.042
C08069=1223.084,-83.976,-37.522,179.632,5.343,149.041
C08070=1223.079,-83.726,-37.533,179.634,5.344,149.040
C08071=1223.074,-83.477,-37.544,179.636,5.343,149.040
C08072=1223.069,-83.227,-37.555,179.639,5.344,149.039
C08073=1223.063,-82.977,-37.567,179.641,5.343,149.038
C08074=1223.059,-82.728,-37.578,179.644,5.344,149.037
C08075=1223.053,-82.478,-37.588,179.646,5.344,149.037
C08076=1223.048,-82.228,-37.600,179.649,5.344,149.036
C08077=1223.043,-81.978,-37.611,179.651,5.344,149.035
C08078=1223.037,-81.729,-37.621,179.653,5.344,149.035
C08079=1223.033,-81.479,-37.633,179.655,5.344,149.034
C08080=1223.027,-81.229,-37.645,179.658,5.344,149.033
C08081=1223.023,-80.980,-37.656,179.660,5.344,149.032
C08082=1223.017,-80.730,-37.666,179.663,5.344,149.032
C08083=1223.012,-80.480,-37.678,179.664,5.344,149.031
C08084=1223.007,-80.231,-37.689,179.667,5.345,149.031
C08085=1223.002,-79.982,-37.700,179.669,5.344,149.030
C08086=1222.996,-79.731,-37.711,179.672,5.345,149.029
C08087=1222.991,-79.482,-37.723,179.674,5.344,149.028
C08088=1222.986,-79.232,-37.734,179.677,5.345,149.028
C08089=1222.980,-78.983,-37.745,179.679,5.345,149.027
C08090=1222.975,-78.732,-37.756,179.681,5.345,149.026
C08091=1222.970,-78.483,-37.768,179.684,5.345,149.026
C08092=1222.965,-78.233,-37.779,179.686,5.345,149.025
C08093=1222.960,-77.984,-37.790,179.689,5.346,149.024
C08094=1222.955,-77.734,-37.802,179.691,5.345,149.023
C08095=1222.950,-77.484,-37.813,179.694,5.346,149.023
C08096=1222.945,-77.234,-37.824,179.696,5.345,149.022
C08097=1222.939,-76.985,-37.835,179.698,5.346,149.021
C08098=1222.934,-76.735,-37.847,179.700,5.345,149.021
C08099=1222.929,-76.485,-37.859,179.703,5.346,149.020
C08100=1222.924,-76.236,-37.870,179.705,5.346,149.019
C08101=1222.918,-75.986,-37.881,179.707,5.346,149.019
C08102=1222.913,-75.736,-37.892,179.709,5.346,149.018
C08103=1222.908,-75.487,-37.903,179.712,5.346,149.017
C08104=1222.903,-75.237,-37.915,179.714,5.346,149.017
C08105=1222.897,-74.966,-37.927,179.717,5.346,149.016
C08106=1222.891,-74.696,-37.940,179.720,5.347,149.015
C08107=1222.886,-74.425,-37.952,179.722,5.346,149.014
C08108=1222.881,-74.156,-37.964,179.725,5.347,149.014
C08109=1222.875,-73.906,-37.976,179.727,5.347,149.013
C08110=1222.870,-73.656,-37.987,179.730,5.347,149.012
C08111=1222.865,-73.406,-37.999,179.732,5.347,149.011
C08112=1222.859,-73.157,-38.009,179.734,5.347,149.011
C08113=1222.854,-72.907,-38.021,179.737,5.347,149.010
C08114=1222.849,-72.657,-38.033,179.739,5.347,149.009
C08115=1222.844,-72.407,-38.045,179.742,5.348,149.009
C08116=1222.839,-72.158,-38.056,179.744,5.347,149.008
C08117=1222.833,-71.908,-38.067,179.746,5.348,149.007
C08118=1222.828,-71.659,-38.079,179.749,5.348,149.006
C08119=1222.823,-71.409,-38.091,179.751,5.348,149.006
C08120=1222.818,-71.159,-38.102,179.754,5.348,149.005
C08121=1222.813,-70.909,-38.114,179.756,5.348,149.005
C08122=1222.807,-70.659,-38.126,179.758,5.349,149.004
C08123=1222.803,-70.410,-38.137,179.760,5.348,149.003
C08124=1222.797,-70.160,-38.148,179.763,5.349,149.002
C08125=1222.792,-69.911,-38.160,179.765,5.348,149.002
C08126=1222.787,-69.661,-38.172,179.768,5.349,149.001
C08127=1222.782,-69.411,-38.183,179.770,5.349,149.000
C08128=1222.776,-69.161,-38.195,179.772,5.349,149.000
C08129=1222.772,-68.912,-38.206,179.775,5.349,148.999
C08130=1222.766,-68.662,-38.218,179.777,5.349,148.998
C08131=1222.760,-68.412,-38.229,179.780,5.350,148.997
C08132=1222.756,-68.163,-38.241,179.782,5.349,148.997
C08133=1222.751,-67.914,-38.253,179.785,5.350,148.996
C08134=1222.746,-67.664,-38.265,179.787,5.349,148.995
C08135=1222.740,-67.414,-38.277,179.789,5.350,148.995
C08136=1222.736,-67.164,-38.288,179.791,5.349,148.994
C08137=1222.730,-66.914,-38.300,179.794,5.350,148.993
C08138=1222.725,-66.664,-38.312,179.797,5.350,148.993
C08139=1222.720,-66.415,-38.323,179.799,5.350,148.992
C08140=1222.714,-66.166,-38.334,179.802,5.351,148.991
C08141=1222.709,-65.916,-38.347,179.804,5.350,148.990
C08142=1222.704,-65.667,-38.358,179.806,5.351,148.990
C08143=1222.699,-65.417,-38.370,179.808,5.350,148.989
C08144=1222.694,-65.167,-38.381,179.811,5.351,148.988
C08145=1222.689,-64.917,-38.393,179.813,5.350,148.988
C08146=1222.683,-64.667,-38.405,179.816,5.351,148.987
C08147=1222.679,-64.418,-38.417,179.818,5.352,148.986
C08148=1222.674,-64.168,-38.429,179.820,5.351,148.986
C08149=1222.668,-63.918,-38.441,179.823,5.352,148.985
C08150=1222.663,-63.669,-38.452,179.825,5.352,148.984
C08151=1222.658,-63.419,-38.464,179.828,5.352,148.984
C08152=1222.653,-63.169,-38.477,179.830,5.352,148.983
C08153=1222.648,-62.920,-38.488,179.832,5.352,148.982
C08154=1222.642,-62.671,-38.500,179.834,5.352,148.981
C08155=1222.637,-62.421,-38.511,179.837,5.352,148.981
C08156=1222.631,-62.171,-38.523,179.840,5.353,148.980
C08157=1222.627,-61.922,-38.535,179.842,5.352,148.979
C08158=1222.621,-61.672,-38.547,179.844,5.353,148.979
C08159=1222.616,-61.422,-38.559,179.847,5.352,148.978
C08160=1222.612,-61.173,-38.571,179.849,5.353,148.977
C08161=1222.606,-60.923,-38.583,179.851,5.353,148.976
C08162=1222.601,-60.673,-38.595,179.854,5.353,148.976
C08163=1222.595,-60.423,-38.607,179.857,5.354,148.975
C08164=1222.591,-60.174,-38.619,179.859,5.353,148.974
C08165=1222.586,-59.924,-38.631,179.861,5.354,148.974
C08166=1222.580,-59.674,-38.643,179.863,5.353,148.973
C08167=1222.575,-59.425,-38.655,179.866,5.354,148.972
C08168=1222.570,-59.175,-38.666,179.868,5.353,148.972
C08169=1222.565,-58.925,-38.678,179.871,5.354,148.971
C08170=1222.560,-58.676,-38.691,179.874,5.354,148.970
C08171=1222.554,-58.426,-38.703,179.876,5.354,148.969
C08172=1222.550,-58.176,-38.714,179.878,5.354,148.969
C08173=1222.544,-57.927,-38.727,179.880,5.354,148.968
C08174=1222.539,-57.677,-38.739,179.883,5.355,148.967
C08175=1222.534,-57.428,-38.751,179.885,5.354,148.967
C08176=1222.529,-57.178,-38.763,179.888,5.355,148.966
C08177=1222.524,-56.928,-38.774,179.891,5.355,148.965
C08178=1222.519,-56.678,-38.787,179.893,5.355,148.965
C08179=1222.514,-56.428,-38.799,179.895,5.355,148.964
C08180=1222.509,-56.179,-38.812,179.897,5.355,148.963
C08181=1222.503,-55.929,-38.824,179.900,5.355,148.962
C08182=1222.499,-55.679,-38.835,179.903,5.356,148.962
C08183=1222.493,-55.430,-38.848,179.904,5.356,148.961
C08184=1222.488,-55.180,-38.859,179.907,5.356,148.961
C08185=1222.483,-54.931,-38.872,179.909,5.356,148.960
C08186=1222.478,-54.681,-38.884,179.912,5.357,148.959
C08187=1222.472,-54.432,-38.897,179.914,5.356,148.958
C08188=1222.468,-54.182,-38.908,179.916,5.357,148.958
C08189=1222.463,-53.933,-38.920,179.919,5.357,148.957
C08190=1222.457,-53.683,-38.932,179.921,5.357,148.956
C08191=1222.452,-53.433,-38.945,179.924,5.357,148.956
C08192=1222.447,-53.183,-38.957,179.926,5.357,148.955
C08193=1222.442,-52.933,-38.970,179.929,5.357,148.954
C08194=1222.437,-52.684,-38.982,179.931,5.358,148.953
C08195=1222.432,-52.434,-38.994,179.933,5.358,148.953
C08196=1222.426,-52.184,-39.006,179.936,5.358,148.952
C08197=1222.422,-51.935,-39.018,179.938,5.358,148.951
C08198=1222.416,-51.685,-39.030,179.941,5.358,148.951
C08199=1222.411,-51.436,-39.043,179.943,5.359,148.950
C08200=1222.406,-51.186,-39.055,179.946,5.358,148.949
C08201=1222.401,-50.937,-39.067,179.948,5.359,148.949
C08202=1222.396,-50.687,-39.080,179.950,5.359,148.948
C08203=1222.391,-50.437,-39.092,179.953,5.359,148.947
C08204=1222.386,-50.187,-39.105,179.956,5.359,148.946
C08205=1222.380,-49.938,-39.116,179.958,5.359,148.946
C08206=1222.375,-49.688,-39.129,179.960,5.360,148.945
C08207=1222.370,-49.439,-39.142,179.962,5.359,148.944
C08208=1222.364,-49.189,-39.154,179.965,5.360,148.944
C08209=1222.359,-48.919,-39.167,179.968,5.360,148.943
C08210=1222.354,-48.649,-39.180,179.970,5.360,148.942
C08211=1222.348,-48.380,-39.194,179.973,5.360,148.941
C08212=1222.342,-48.109,-39.207,179.976,5.360,148.941
C08213=1222.337,-47.860,-39.220,179.978,5.360,148.940
C08214=1222.332,-47.611,-39.232,179.980,5.361,148.939
C08215=1222.327,-47.361,-39.244,179.983,5.361,148.938
C08216=1222.322,-47.111,-39.257,179.985,5.361,148.938
C08217=1222.317,-46.861,-39.270,179.988,5.361,148.937
C08218=1222.312,-46.611,-39.282,179.991,5.362,148.936
C08219=1222.307,-46.362,-39.294,179.993,5.361,148.936
C08220=1222.301,-46.113,-39.307,179.995,5.362,148.935
C08221=1222.296,-45.863,-39.319,179.997,5.362,148.934
C08222=1222.291,-45.613,-39.332,-180.000,5.362,148.934
C08223=1222.286,-45.363,-39.344,-179.997,5.362,148.933
C08224=1222.281,-45.114,-39.357,-179.995,5.362,148.932
C08225=1222.276,-44.864,-39.369,-179.993,5.363,148.931
C08226=1222.271,-44.615,-39.381,-179.990,5.362,148.931
C08227=1222.266,-44.365,-39.394,-179.988,5.363,148.930
C08228=1222.261,-44.116,-39.407,-179.985,5.363,148.929
C08229=1222.255,-43.866,-39.420,-179.983,5.363,148.929
C08230=1222.250,-43.616,-39.432,-179.980,5.363,148.928
C08231=1222.245,-43.367,-39.445,-179.978,5.363,148.927
C08232=1222.240,-43.117,-39.458,-179.976,5.364,148.927
C08233=1222.235,-42.867,-39.470,-179.973,5.364,148.926
C08234=1222.230,-42.618,-39.483,-179.971,5.364,148.925
C08235=1222.224,-42.368,-39.495,-179.969,5.365,148.925
C08236=1222.220,-42.118,-39.508,-179.966,5.365,148.924
C08237=1222.215,-41.869,-39.520,-179.964,5.365,148.923
C08238=1222.209,-41.619,-39.533,-179.961,5.365,148.923
C08239=1222.204,-41.370,-39.546,-179.959,5.365,148.922
C08240=1222.199,-41.120,-39.559,-179.957,5.365,148.921
C08241=1222.194,-40.870,-39.571,-179.954,5.366,148.920
C08242=1222.189,-40.621,-39.583,-179.952,5.366,148.920
C08243=1222.184,-40.371,-39.596,-179.949,5.366,148.919
C08244=1222.179,-40.121,-39.609,-179.946,5.367,148.918
C08245=1222.173,-39.872,-39.622,-179.944,5.366,148.918
C08246=1222.168,-39.622,-39.635,-179.942,5.367,148.917
C08247=1222.163,-39.373,-39.647,-179.940,5.366,148.916
C08248=1222.158,-39.123,-39.660,-179.937,5.367,148.916
C08249=1222.153,-38.874,-39.673,-179.934,5.367,148.915
C08250=1222.148,-38.624,-39.686,-179.932,5.367,148.914
C08251=1222.143,-38.373,-39.698,-179.930,5.367,148.913
C08252=1222.138,-38.124,-39.711,-179.927,5.368,148.913
C08253=1222.132,-37.875,-39.724,-179.925,5.368,148.912
C08254=1222.127,-37.625,-39.736,-179.922,5.368,148.911
C08255=1222.122,-37.375,-39.750,-179.920,5.369,148.911
C08256=1222.117,-37.126,-39.762,-179.917,5.368,148.910
C08257=1222.112,-36.876,-39.775,-179.915,5.369,148.909
C08258=1222.107,-36.626,-39.788,-179.913,5.368,148.909
C08259=1222.102,-36.377,-39.801,-179.910,5.369,148.908
C08260=1222.096,-36.127,-39.814,-179.907,5.369,148.907
C08261=1222.092,-35.877,-39.827,-179.905,5.369,148.906
C08262=1222.087,-35.628,-39.839,-179.903,5.370,148.906
C08263=1222.081,-35.379,-39.852,-179.900,5.370,148.905
C08264=1222.076,-35.128,-39.866,-179.898,5.370,148.904
C08265=1222.071,-34.879,-39.878,-179.895,5.370,148.904
C08266=1222.066,-34.630,-39.891,-179.893,5.371,148.903
C08267=1222.061,-34.379,-39.904,-179.890,5.370,148.902
C08268=1222.056,-34.130,-39.917,-179.888,5.371,148.902
C08269=1222.051,-33.881,-39.930,-179.886,5.371,148.901
C08270=1222.046,-33.631,-39.943,-179.883,5.371,148.900
C08271=1222.040,-33.382,-39.956,-179.880,5.372,148.899
C08272=1222.035,-33.133,-39.969,-179.878,5.371,148.899
C08273=1222.031,-32.882,-39.982,-179.876,5.372,148.898
C08274=1222.025,-32.633,-39.995,-179.873,5.372,148.897
C08275=1222.020,-32.383,-40.008,-179.871,5.372,148.897
C08276=1222.015,-32.134,-40.021,-179.868,5.372,148.896
C08277=1222.009,-31.884,-40.034,-179.866,5.373,148.895
C08278=1222.005,-31.634,-40.047,-179.863,5.373,148.895
C08279=1222.000,-31.385,-40.060,-179.861,5.373,148.894
C08280=1221.994,-31.136,-40.073,-179.858,5.374,148.893
C08281=1221.990,-30.886,-40.086,-179.856,5.373,148.892
C08282=1221.985,-30.636,-40.099,-179.853,5.374,148.892
C08283=1221.979,-30.386,-40.113,-179.851,5.374,148.891
C08284=1221.974,-30.137,-40.125,-179.849,5.374,148.890
C08285=1221.969,-29.888,-40.139,-179.846,5.374,148.890
C08286=1221.964,-29.638,-40.152,-179.843,5.375,148.889
C08287=1221.959,-29.388,-40.165,-179.841,5.375,148.888
C08288=1221.954,-29.138,-40.178,-179.839,5.375,148.888
C08289=1221.949,-28.889,-40.191,-179.836,5.376,148.887
C08290=1221.944,-28.639,-40.204,-179.834,5.375,148.886
C08291=1221.938,-28.390,-40.218,-179.831,5.376,148.886
C08292=1221.933,-28.140,-40.230,-179.829,5.376,148.885
C08293=1221.928,-27.890,-40.244,-179.826,5.376,148.884
C08294=1221.923,-27.641,-40.257,-179.824,5.376,148.883
C08295=1221.918,-27.391,-40.271,-179.821,5.377,148.883
C08296=1221.913,-27.142,-40.283,-179.819,5.377,148.882
C08297=1221.908,-26.892,-40.296,-179.816,5.377,148.881
C08298=1221.903,-26.643,-40.310,-179.814,5.378,148.881
C08299=1221.898,-26.393,-40.323,-179.812,5.377,148.880
C08300=1221.892,-26.143,-40.336,-179.810,5.378,148.879
C08301=1221.888,-25.894,-40.350,-179.807,5.379,148.879
C08302=1221.882,-25.644,-40.363,-179.805,5.378,148.878
C08303=1221.877,-25.395,-40.376,-179.802,5.379,148.877
C08304=1221.872,-25.145,-40.390,-179.799,5.379,148.877
C08305=1221.867,-24.896,-40.403,-179.797,5.379,148.876
C08306=1221.862,-24.645,-40.416,-179.795,5.379,148.875
C08307=1221.857,-24.396,-40.430,-179.792,5.380,148.875
C08308=1221.852,-24.146,-40.443,-179.790,5.380,148.874
C08309=1221.847,-23.897,-40.456,-179.787,5.380,148.873
C08310=1221.842,-23.647,-40.470,-179.785,5.381,148.873
C08311=1221.837,-23.398,-40.483,-179.783,5.380,148.872
C08312=1221.832,-23.148,-40.497,-179.780,5.381,148.871
C08313=1221.827,-22.878,-40.511,-179.777,5.381,148.870
C08314=1221.821,-22.610,-40.525,-179.774,5.381,148.869
C08315=1221.815,-22.340,-40.539,-179.772,5.381,148.869
C08316=1221.810,-22.071,-40.554,-179.769,5.382,148.868
C08317=1221.805,-21.822,-40.568,-179.767,5.382,148.867
C08318=1221.800,-21.571,-40.581,-179.764,5.383,148.867
C08319=1221.794,-21.322,-40.594,-179.762,5.382,148.866
C08320=1221.789,-21.072,-40.608,-179.759,5.383,148.865
C08321=1221.784,-20.823,-40.621,-179.757,5.383,148.865
C08322=1221.779,-20.573,-40.635,-179.755,5.383,148.864
C08323=1221.774,-20.324,-40.648,-179.752,5.383,148.863
C08324=1221.769,-20.074,-40.662,-179.749,5.384,148.863
C08325=1221.764,-19.824,-40.676,-179.747,5.384,148.862
C08326=1221.759,-19.575,-40.689,-179.744,5.384,148.861
C08327=1221.754,-19.325,-40.702,-179.742,5.385,148.860
C08328=1221.749,-19.076,-40.716,-179.739,5.385,148.860
C08329=1221.744,-18.826,-40.729,-179.737,5.385,148.859
C08330=1221.738,-18.577,-40.743,-179.734,5.385,148.858
C08331=1221.734,-18.327,-40.756,-179.732,5.386,148.858
C08332=1221.729,-18.077,-40.770,-179.730,5.386,148.857
C08333=1221.724,-17.828,-40.783,-179.727,5.386,148.856
C08334=1221.719,-17.578,-40.797,-179.724,5.387,148.856
C08335=1221.713,-17.329,-40.811,-179.722,5.386,148.855
C08336=1221.709,-17.079,-40.824,-179.720,5.387,148.854
C08337=1221.703,-16.830,-40.838,-179.717,5.387,148.854
C08338=1221.698,-16.580,-40.852,-179.714,5.388,148.853
C08339=1221.693,-16.330,-40.865,-179.712,5.387,148.852
C08340=1221.688,-16.081,-40.879,-179.710,5.388,148.851
C08341=1221.683,-15.831,-40.893,-179.707,5.388,148.851
C08342=1221.678,-15.582,-40.906,-179.705,5.388,148.850
C08343=1221.673,-15.332,-40.920,-179.702,5.389,148.849
C08344=1221.668,-15.082,-40.934,-179.700,5.389,148.849
C08345=1221.662,-14.833,-40.948,-179.697,5.390,148.848
C08346=1221.658,-14.583,-40.961,-179.695,5.389,148.847
C08347=1221.653,-14.333,-40.975,-179.692,5.390,148.847
C08348=1221.647,-14.084,-40.989,-179.689,5.390,148.846
C08349=1221.643,-13.834,-41.002,-179.688,5.390,148.845
C08350=1221.637,-13.585,-41.016,-179.685,5.391,148.845
C08351=1221.632,-13.336,-41.030,-179.683,5.391,148.844
C08352=1221.627,-13.085,-41.044,-179.681,5.391,148.843
C08353=1221.622,-12.837,-41.057,-179.678,5.392,148.843
C08354=1221.617,-12.587,-41.071,-179.675,5.392,148.842
C08355=1221.612,-12.337,-41.086,-179.673,5.393,148.841
C08356=1221.606,-12.088,-41.099,-179.670,5.392,148.841
C08357=1221.602,-11.838,-41.112,-179.668,5.393,148.840
C08358=1221.597,-11.588,-41.127,-179.665,5.393,148.839
C08359=1221.591,-11.339,-41.140,-179.662,5.394,148.838
C08360=1221.586,-11.089,-41.154,-179.660,5.394,148.838
C08361=1221.582,-10.840,-41.168,-179.658,5.394,148.837
C08362=1221.576,-10.591,-41.182,-179.655,5.395,148.836
C08363=1221.571,-10.341,-41.196,-179.653,5.394,148.836
C08364=1221.566,-10.091,-41.210,-179.650,5.395,148.835
C08365=1221.561,-9.842,-41.224,-179.648,5.395,148.834
C08366=1221.556,-9.592,-41.237,-179.645,5.396,148.834
C08367=1221.551,-9.343,-41.252,-179.643,5.395,148.833
C08368=1221.546,-9.093,-41.266,-179.640,5.396,148.832
C08369=1221.541,-8.843,-41.279,-179.638,5.396,148.832
C08370=1221.536,-8.593,-41.293,-179.635,5.397,148.831
C08371=1221.531,-8.344,-41.308,-179.633,5.397,148.830
C08372=1221.526,-8.095,-41.321,-179.630,5.397,148.829
C08373=1221.521,-7.845,-41.335,-179.628,5.398,148.829
C08374=1221.516,-7.596,-41.349,-179.626,5.397,148.828
C08375=1221.511,-7.346,-41.364,-179.623,5.398,148.827
C08376=1221.505,-7.096,-41.377,-179.620,5.398,148.827
C08377=1221.500,-6.847,-41.391,-179.618,5.399,148.826
C08378=1221.495,-6.597,-41.405,-179.616,5.399,148.825
C08379=1221.491,-6.347,-41.419,-179.613,5.399,148.825
C08380=1221.485,-6.098,-41.433,-179.610,5.400,148.824
C08381=1221.481,-5.849,-41.447,-179.608,5.400,148.823
C08382=1221.476,-5.599,-41.462,-179.605,5.400,148.823
C08383=1221.471,-5.349,-41.476,-179.603,5.400,148.822
C08384=1221.465,-5.100,-41.490,-179.601,5.401,148.821
C08385=1221.460,-4.851,-41.504,-179.598,5.402,148.821
C08386=1221.455,-4.601,-41.518,-179.596,5.401,148.820
C08387=1221.450,-4.351,-41.533,-179.593,5.402,148.819
C08388=1221.445,-4.102,-41.547,-179.591,5.403,148.819
C08389=1221.440,-3.852,-41.561,-179.588,5.403,148.818
C08390=1221.435,-3.603,-41.575,-179.586,5.403,148.817
C08391=1221.431,-3.353,-41.589,-179.583,5.403,148.817
C08392=1221.426,-3.104,-41.603,-179.581,5.404,148.816
C08393=1221.420,-2.855,-41.617,-179.578,5.404,148.815
C08394=1221.415,-2.605,-41.631,-179.576,5.404,148.815
C08395=1221.410,-2.355,-41.646,-179.573,5.404,148.814
C08396=1221.405,-2.106,-41.660,-179.571,5.405,148.813
C08397=1221.400,-1.856,-41.674,-179.568,5.406,148.812
C08398=1221.395,-1.607,-41.688,-179.566,5.405,148.812
C08399=1221.390,-1.357,-41.702,-179.563,5.406,148.811
C08400=1221.385,-1.107,-41.717,-179.560,5.406,148.810
C08401=1221.380,-0.858,-41.731,-179.558,5.407,148.810
C08402=1221.375,-0.608,-41.745,-179.556,5.406,148.809
C08403=1221.370,-0.358,-41.759,-179.553,5.407,148.808
C08404=1221.364,-0.109,-41.773,-179.550,5.408,148.808
C08405=1221.359,0.140,-41.788,-179.548,5.408,148.807
C08406=1221.354,0.390,-41.802,-179.546,5.408,148.806
C08407=1221.350,0.639,-41.817,-179.543,5.408,148.806
C08408=1221.345,0.889,-41.831,-179.540,5.409,148.805
C08409=1221.340,1.139,-41.845,-179.538,5.409,148.804
C08410=1221.334,1.388,-41.860,-179.536,5.410,148.804
C08411=1221.329,1.638,-41.874,-179.534,5.410,148.803
C08412=1221.324,1.887,-41.888,-179.531,5.410,148.802
C08413=1221.319,2.137,-41.903,-179.528,5.411,148.802
C08414=1221.314,2.386,-41.918,-179.526,5.411,148.801
C08415=1221.309,2.636,-41.932,-179.524,5.411,148.800
C08416=1221.304,2.886,-41.946,-179.521,5.412,148.800
C08417=1221.299,3.154,-41.962,-179.518,5.412,148.799
C08418=1221.293,3.423,-41.977,-179.515,5.412,148.798
C08419=1221.287,3.692,-41.993,-179.512,5.413,148.797
C08420=1221.282,3.961,-42.009,-179.510,5.413,148.797
C08421=1221.277,4.211,-42.023,-179.507,5.414,148.796
C08422=1221.272,4.460,-42.037,-179.505,5.414,148.795
C08423=1221.267,4.710,-42.052,-179.502,5.414,148.795
C08424=1221.262,4.959,-42.066,-179.500,5.415,148.794
C08425=1221.258,5.209,-42.081,-179.497,5.415,148.793
C08426=1221.252,5.459,-42.096,-179.494,5.416,148.792
C08427=1221.247,5.708,-42.111,-179.492,5.415,148.792
C08428=1221.242,5.957,-42.124,-179.490,5.416,148.791
C08429=1221.237,6.207,-42.139,-179.487,5.416,148.790
C08430=1221.232,6.457,-42.153,-179.485,5.417,148.790
C08431=1221.227,6.706,-42.168,-179.483,5.417,148.789
C08432=1221.222,6.955,-42.182,-179.480,5.418,148.789
C08433=1221.216,7.205,-42.197,-179.477,5.418,148.788
C08434=1221.212,7.454,-42.212,-179.475,5.419,148.787
C08435=1221.207,7.704,-42.226,-179.472,5.419,148.787
C08436=1221.202,7.954,-42.241,-179.470,5.419,148.786
C08437=1221.197,8.203,-42.256,-179.467,5.419,148.785
C08438=1221.191,8.453,-42.271,-179.465,5.420,148.784
C08439=1221.187,8.702,-42.286,-179.462,5.420,148.784
C08440=1221.182,8.952,-42.300,-179.460,5.421,148.783
C08441=1221.177,9.202,-42.314,-179.457,5.421,148.782
C08442=1221.172,9.451,-42.330,-179.455,5.421,148.782
C08443=1221.167,9.701,-42.344,-179.452,5.422,148.781
C08444=1221.162,9.950,-42.359,-179.449,5.422,148.780
C08445=1221.157,10.199,-42.373,-179.447,5.423,148.780
C08446=1221.151,10.449,-42.388,-179.445,5.422,148.779
C08447=1221.147,10.699,-42.403,-179.442,5.423,148.778
C08448=1221.142,10.948,-42.417,-179.440,5.424,148.778
C08449=1221.137,11.197,-42.432,-179.437,5.424,148.777
C08450=1221.131,11.447,-42.447,-179.435,5.425,148.776
C08451=1221.127,11.696,-42.462,-179.433,5.425,148.776
C08452=1221.122,11.946,-42.477,-179.430,5.425,148.775
C08453=1221.117,12.195,-42.492,-179.427,5.426,148.774
C08454=1221.111,12.445,-42.506,-179.425,5.426,148.774
C08455=1221.107,12.694,-42.521,-179.422,5.427,148.773
C08456=1221.102,12.944,-42.536,-179.419,5.427,148.772
C08457=1221.096,13.193,-42.551,-179.417,5.427,148.772
C08458=1221.091,13.443,-42.566,-179.415,5.428,148.771
C08459=1221.087,13.692,-42.581,-179.412,5.428,148.770
C08460=1221.081,13.942,-42.595,-179.409,5.429,148.770
C08461=1221.076,14.191,-42.610,-179.407,5.429,148.769
C08462=1221.072,14.441,-42.625,-179.405,5.429,148.768
C08463=1221.066,14.691,-42.640,-179.402,5.429,148.768
C08464=1221.061,14.940,-42.655,-179.400,5.430,148.767
C08465=1221.057,15.189,-42.670,-179.397,5.431,148.766
C08466=1221.051,15.439,-42.685,-179.394,5.431,148.766
C08467=1221.046,15.688,-42.699,-179.392,5.432,148.765
C08468=1221.041,15.938,-42.715,-179.390,5.432,148.764
C08469=1221.036,16.187,-42.730,-179.387,5.432,148.764
C08470=1221.031,16.437,-42.744,-179.384,5.433,148.763
C08471=1221.026,16.687,-42.760,-179.382,5.433,148.762
C08472=1221.021,16.936,-42.775,-179.379,5.434,148.762
C08473=1221.016,17.186,-42.790,-179.377,5.434,148.761
C08474=1221.011,17.435,-42.805,-179.374,5.434,148.760
C08475=1221.006,17.685,-42.819,-179.372,5.434,148.760
C08476=1221.001,17.934,-42.835,-179.369,5.435,148.759
C08477=1220.996,18.183,-42.850,-179.367,5.436,148.758
C08478=1220.991,18.433,-42.865,-179.364,5.436,148.758
C08479=1220.986,18.682,-42.880,-179.362,5.437,148.757
C08480=1220.981,18.932,-42.895,-179.360,5.437,148.756
C08481=1220.976,19.182,-42.910,-179.357,5.437,148.756
C08482=1220.972,19.431,-42.925,-179.354,5.438,148.755
C08483=1220.966,19.681,-42.941,-179.352,5.438,148.754
C08484=1220.962,19.930,-42.956,-179.349,5.439,148.754
C08485=1220.956,20.180,-42.970,-179.346,5.439,148.753
C08486=1220.951,20.429,-42.985,-179.344,5.439,148.752
C08487=1220.946,20.678,-43.001,-179.342,5.440,148.752
C08488=1220.941,20.927,-43.016,-179.339,5.440,148.751
C08489=1220.936,21.178,-43.031,-179.336,5.441,148.750
C08490=1220.932,21.427,-43.046,-179.334,5.441,148.750
C08491=1220.926,21.676,-43.062,-179.332,5.442,148.749
C08492=1220.922,21.926,-43.077,-179.329,5.443,148.748
C08493=1220.916,22.175,-43.092,-179.327,5.442,148.748
C08494=1220.911,22.425,-43.107,-179.324,5.443,148.747
C08495=1220.906,22.675,-43.123,-179.322,5.443,148.746
C08496=1220.902,22.924,-43.138,-179.319,5.444,148.746
C08497=1220.896,23.173,-43.153,-179.316,5.444,148.745
C08498=1220.891,23.423,-43.169,-179.314,5.445,148.744
C08499=1220.886,23.672,-43.184,-179.311,5.446,148.744
C08500=1220.881,23.922,-43.199,-179.309,5.445,148.743
C08501=1220.877,24.172,-43.214,-179.306,5.446,148.742
C08502=1220.871,24.421,-43.230,-179.304,5.446,148.742
C08503=1220.867,24.670,-43.245,-179.301,5.447,148.741
C08504=1220.861,24.919,-43.260,-179.299,5.448,148.741
C08505=1220.856,25.169,-43.276,-179.296,5.448,148.740
C08506=1220.852,25.419,-43.291,-179.294,5.449,148.739
C08507=1220.846,25.668,-43.307,-179.291,5.449,148.738
C08508=1220.842,25.917,-43.322,-179.289,5.449,148.738
C08509=1220.836,26.167,-43.337,-179.286,5.450,148.737
C08510=1220.832,26.417,-43.353,-179.284,5.450,148.736
C08511=1220.827,26.666,-43.368,-179.281,5.451,148.736
C08512=1220.821,26.916,-43.383,-179.278,5.451,148.735
C08513=1220.817,27.165,-43.398,-179.276,5.452,148.734
C08514=1220.811,27.414,-43.414,-179.273,5.453,148.734
C08515=1220.806,27.664,-43.430,-179.271,5.452,148.733
C08516=1220.802,27.913,-43.445,-179.269,5.453,148.733
C08517=1220.796,28.163,-43.460,-179.266,5.454,148.732
C08518=1220.791,28.412,-43.476,-179.263,5.454,148.731
C08519=1220.787,28.662,-43.491,-179.261,5.455,148.731
C08520=1220.781,28.911,-43.507,-179.258,5.455,148.730
C08521=1220.776,29.180,-43.524,-179.256,5.456,148.729
C08522=1220.770,29.448,-43.541,-179.253,5.456,148.729
C08523=1220.766,29.717,-43.557,-179.250,5.457,148.728
C08524=1220.760,29.986,-43.574,-179.248,5.457,148.727
C08525=1220.755,30.236,-43.590,-179.245,5.458,148.727
C08526=1220.751,30.484,-43.605,-179.242,5.458,148.726
C08527=1220.745,30.734,-43.621,-179.240,5.459,148.725
C08528=1220.740,30.984,-43.637,-179.238,5.459,148.724
C08529=1220.735,31.233,-43.652,-179.235,5.459,148.724
C08530=1220.730,31.482,-43.667,-179.232,5.460,148.723
C08531=1220.726,31.732,-43.683,-179.230,5.460,148.722
C08532=1220.720,31.982,-43.699,-179.227,5.461,148.722
C08533=1220.715,32.231,-43.715,-179.225,5.462,148.721
C08534=1220.710,32.480,-43.730,-179.222,5.462,148.721
C08535=1220.706,32.730,-43.746,-179.220,5.463,148.720
C08536=1220.700,32.979,-43.762,-179.217,5.463,148.719
C08537=1220.695,33.229,-43.777,-179.214,5.464,148.719
C08538=1220.691,33.478,-43.793,-179.212,5.464,148.718
C08539=1220.685,33.728,-43.808,-179.210,5.464,148.717
C08540=1220.680,33.977,-43.824,-179.207,5.465,148.717
C08541=1220.676,34.227,-43.841,-179.205,5.466,148.716
C08542=1220.670,34.476,-43.856,-179.202,5.466,148.715
C08543=1220.666,34.725,-43.871,-179.199,5.467,148.715
C08544=1220.661,34.975,-43.887,-179.197,5.467,148.714
C08545=1220.656,35.224,-43.903,-179.194,5.468,148.713
C08546=1220.651,35.474,-43.919,-179.192,5.468,148.713
C08547=1220.646,35.724,-43.935,-179.189,5.469,148.712
C08548=1220.640,35.973,-43.951,-179.186,5.469,148.711
C08549=1220.636,36.222,-43.967,-179.184,5.469,148.711
C08550=1220.631,36.472,-43.982,-179.182,5.470,148.710
C08551=1220.626,36.721,-43.998,-179.179,5.471,148.710
C08552=1220.621,36.971,-44.014,-179.177,5.471,148.709
C08553=1220.616,37.220,-44.030,-179.174,5.472,148.708
C08554=1220.611,37.470,-44.046,-179.171,5.472,148.708
C08555=1220.606,37.719,-44.062,-179.169,5.473,148.707
C08556=1220.601,37.968,-44.077,-179.166,5.473,148.706
C08557=1220.596,38.218,-44.093,-179.164,5.474,148.706
C08558=1220.591,38.467,-44.109,-179.161,5.475,148.705
C08559=1220.587,38.717,-44.125,-179.159,5.475,148.704
C08560=1220.581,38.966,-44.141,-179.156,5.476,148.704
C08561=1220.576,39.216,-44.157,-179.154,5.476,148.703
C08562=1220.571,39.465,-44.173,-179.151,5.476,148.702
C08563=1220.566,39.714,-44.189,-179.149,5.477,148.702
C08564=1220.561,39.965,-44.205,-179.146,5.477,148.701
C08565=1220.556,40.213,-44.221,-179.144,5.478,148.700
C08566=1220.551,40.463,-44.237,-179.141,5.479,148.700
C08567=1220.546,40.712,-44.253,-179.139,5.479,148.699
C08568=1220.541,40.962,-44.269,-179.136,5.480,148.699
C08569=1220.536,41.211,-44.286,-179.133,5.480,148.698
C08570=1220.532,41.460,-44.301,-179.131,5.481,148.697
C08571=1220.527,41.710,-44.317,-179.128,5.482,148.697
C08572=1220.522,41.959,-44.333,-179.126,5.482,148.696
C08573=1220.517,42.209,-44.349,-179.123,5.483,148.695
C08574=1220.512,42.458,-44.365,-179.121,5.484,148.695
C08575=1220.507,42.708,-44.381,-179.118,5.484,148.694
C08576=1220.502,42.957,-44.397,-179.115,5.485,148.693
C08577=1220.497,43.206,-44.413,-179.113,5.484,148.693
C08578=1220.492,43.456,-44.430,-179.111,5.485,148.692
C08579=1220.487,43.705,-44.445,-179.108,5.486,148.691
C08580=1220.482,43.955,-44.462,-179.106,5.486,148.691
C08581=1220.476,44.204,-44.478,-179.103,5.487,148.690
C08582=1220.472,44.454,-44.495,-179.101,5.488,148.690
C08583=1220.466,44.703,-44.510,-179.098,5.488,148.689
C08584=1220.462,44.953,-44.527,-179.095,5.489,148.688
C08585=1220.457,45.202,-44.543,-179.093,5.489,148.688
C08586=1220.452,45.452,-44.559,-179.090,5.490,148.687
C08587=1220.447,45.700,-44.576,-179.088,5.491,148.687
C08588=1220.442,45.951,-44.592,-179.085,5.491,148.686
C08589=1220.437,46.199,-44.608,-179.083,5.492,148.685
C08590=1220.432,46.449,-44.624,-179.080,5.492,148.684
C08591=1220.428,46.699,-44.641,-179.077,5.493,148.684
C08592=1220.423,46.948,-44.657,-179.075,5.493,148.683
C08593=1220.418,47.198,-44.673,-179.072,5.494,148.682
C08594=1220.413,47.447,-44.689,-179.070,5.495,148.682
C08595=1220.408,47.696,-44.706,-179.067,5.496,148.681
C08596=1220.402,47.946,-44.722,-179.065,5.496,148.681
C08597=1220.398,48.195,-44.739,-179.062,5.497,148.680
C08598=1220.393,48.444,-44.755,-179.059,5.497,148.679
C08599=1220.388,48.694,-44.771,-179.057,5.498,148.679
C08600=1220.383,48.943,-44.787,-179.055,5.499,148.678
C08601=1220.378,49.192,-44.804,-179.052,5.499,148.678
C08602=1220.374,49.442,-44.820,-179.050,5.499,148.677
C08603=1220.368,49.692,-44.837,-179.047,5.500,148.676
C08604=1220.363,49.941,-44.853,-179.045,5.500,148.676
C08605=1220.358,50.190,-44.870,-179.042,5.501,148.675
C08606=1220.353,50.440,-44.886,-179.040,5.502,148.674
C08607=1220.349,50.689,-44.902,-179.037,5.502,148.674
C08608=1220.344,50.938,-44.919,-179.035,5.503,148.673
C08609=1220.339,51.188,-44.936,-179.032,5.503,148.672
C08610=1220.333,51.437,-44.951,-179.029,5.504,148.672
C08611=1220.329,51.687,-44.968,-179.027,5.504,148.671
C08612=1220.324,51.936,-44.985,-179.025,5.505,148.671
C08613=1220.319,52.185,-45.001,-179.022,5.506,148.670
C08614=1220.314,52.435,-45.018,-179.019,5.506,148.669
C08615=1220.309,52.684,-45.034,-179.017,5.507,148.669
C08616=1220.304,52.934,-45.051,-179.014,5.508,148.668
C08617=1220.300,53.183,-45.067,-179.011,5.508,148.667
C08618=1220.294,53.432,-45.084,-179.009,5.509,148.667
C08619=1220.289,53.682,-45.101,-179.007,5.510,148.666
C08620=1220.285,53.931,-45.118,-179.004,5.510,148.666
C08621=1220.279,54.181,-45.133,-179.001,5.511,148.665
C08622=1220.274,54.431,-45.150,-178.999,5.511,148.664
C08623=1220.270,54.680,-45.167,-178.996,5.512,148.664
C08624=1220.265,54.929,-45.183,-178.994,5.513,148.663
C08625=1220.259,55.198,-45.202,-178.991,5.513,148.662
C08626=1220.254,55.466,-45.220,-178.988,5.515,148.662
C08627=1220.249,55.735,-45.237,-178.985,5.515,148.661
C08628=1220.243,56.003,-45.255,-178.983,5.516,148.660
C08629=1220.239,56.252,-45.272,-178.980,5.516,148.660
C08630=1220.234,56.501,-45.288,-178.978,5.517,148.659
C08631=1220.228,56.751,-45.306,-178.975,5.517,148.658
C08632=1220.224,57.000,-45.322,-178.972,5.518,148.658
C08633=1220.219,57.249,-45.339,-178.970,5.519,148.657
C08634=1220.214,57.499,-45.356,-178.968,5.520,148.657
C08635=1220.209,57.749,-45.373,-178.965,5.520,148.656
C08636=1220.205,57.998,-45.389,-178.962,5.521,148.655
C08637=1220.199,58.247,-45.406,-178.960,5.521,148.655
C08638=1220.194,58.497,-45.423,-178.957,5.522,148.654
C08639=1220.190,58.746,-45.440,-178.955,5.523,148.654
C08640=1220.184,58.995,-45.456,-178.952,5.523,148.653
C08641=1220.179,59.245,-45.473,-178.950,5.524,148.652
C08642=1220.174,59.494,-45.490,-178.947,5.524,148.652
C08643=1220.170,59.744,-45.507,-178.944,5.525,148.651
C08644=1220.165,59.993,-45.523,-178.942,5.526,148.650
C08645=1220.159,60.243,-45.541,-178.940,5.526,148.650
C08646=1220.155,60.492,-45.557,-178.937,5.527,148.649
C08647=1220.150,60.742,-45.575,-178.934,5.528,148.648
C08648=1220.145,60.991,-45.591,-178.932,5.528,148.648
C08649=1220.141,61.239,-45.608,-178.929,5.529,148.647
C08650=1220.135,61.489,-45.625,-178.927,5.530,148.647
C08651=1220.131,61.739,-45.642,-178.924,5.530,148.646
C08652=1220.125,61.988,-45.659,-178.922,5.531,148.645
C08653=1220.121,62.237,-45.676,-178.919,5.531,148.645
C08654=1220.115,62.487,-45.693,-178.917,5.532,148.644
C08655=1220.111,62.737,-45.710,-178.914,5.534,148.644
C08656=1220.105,62.985,-45.727,-178.911,5.534,148.643
C08657=1220.101,63.235,-45.744,-178.908,5.535,148.642
C08658=1220.096,63.484,-45.761,-178.906,5.535,148.642
C08659=1220.091,63.734,-45.778,-178.904,5.536,148.641
C08660=1220.086,63.984,-45.795,-178.901,5.537,148.641
C08661=1220.081,64.232,-45.811,-178.898,5.537,148.640
C08662=1220.076,64.482,-45.829,-178.896,5.538,148.639
C08663=1220.071,64.731,-45.846,-178.894,5.539,148.639
C08664=1220.066,64.981,-45.863,-178.891,5.540,148.638
C08665=1220.062,65.230,-45.880,-178.888,5.540,148.637
C08666=1220.056,65.479,-45.898,-178.886,5.541,148.637
C08667=1220.052,65.728,-45.914,-178.883,5.541,148.636
C08668=1220.047,65.978,-45.932,-178.881,5.542,148.636
C08669=1220.042,66.228,-45.948,-178.878,5.543,148.635
C08670=1220.037,66.477,-45.966,-178.876,5.543,148.634
C08671=1220.033,66.726,-45.983,-178.873,5.544,148.634
C08672=1220.027,66.975,-46.000,-178.871,5.545,148.633
C08673=1220.022,67.225,-46.018,-178.868,5.545,148.633
C08674=1220.017,67.474,-46.034,-178.866,5.546,148.632
C08675=1220.012,67.724,-46.052,-178.862,5.547,148.631
C08676=1220.008,67.973,-46.069,-178.860,5.548,148.631
C08677=1220.003,68.222,-46.086,-178.858,5.549,148.630
C08678=1219.998,68.472,-46.104,-178.855,5.549,148.630
C08679=1219.993,68.721,-46.121,-178.852,5.550,148.629
C08680=1219.988,68.970,-46.138,-178.850,5.551,148.628
C08681=1219.983,69.219,-46.155,-178.848,5.552,148.628
C08682=1219.978,69.469,-46.173,-178.845,5.552,148.627
C08683=1219.973,69.719,-46.190,-178.842,5.553,148.626
C08684=1219.969,69.968,-46.207,-178.840,5.553,148.626
C08685=1219.964,70.217,-46.224,-178.838,5.554,148.625
C08686=1219.959,70.466,-46.242,-178.835,5.555,148.625
C08687=1219.954,70.716,-46.259,-178.832,5.555,148.624
C08688=1219.949,70.966,-46.276,-178.829,5.557,148.623
C08689=1219.944,71.214,-46.294,-178.827,5.558,148.623
C08690=1219.939,71.464,-46.311,-178.824,5.558,148.622
C08691=1219.934,71.713,-46.329,-178.822,5.559,148.622
C08692=1219.929,71.963,-46.346,-178.819,5.559,148.621
C08693=1219.925,72.212,-46.363,-178.816,5.560,148.620
C08694=1219.920,72.461,-46.381,-178.814,5.561,148.620
C08695=1219.915,72.711,-46.399,-178.812,5.561,148.619
C08696=1219.910,72.960,-46.415,-178.809,5.562,148.619
C08697=1219.905,73.209,-46.433,-178.806,5.563,148.618
C08698=1219.900,73.459,-46.450,-178.804,5.564,148.617
C08699=1219.895,73.708,-46.468,-178.802,5.564,148.617
C08700=1219.891,73.958,-46.485,-178.798,5.566,148.616
C08701=1219.886,74.207,-46.503,-178.796,5.566,148.616
C08702=1219.881,74.456,-46.521,-178.794,5.567,148.615
C08703=1219.876,74.706,-46.538,-178.791,5.568,148.614
C08704=1219.871,74.955,-46.556,-178.788,5.568,148.614
C08705=1219.866,75.204,-46.573,-178.786,5.569,148.613
C08706=1219.861,75.453,-46.591,-178.784,5.570,148.613
C08707=1219.856,75.702,-46.609,-178.781,5.570,148.612
C08708=1219.851,75.952,-46.626,-178.778,5.571,148.611
C08709=1219.846,76.201,-46.643,-178.776,5.573,148.611
C08710=1219.841,76.451,-46.660,-178.773,5.573,148.610
C08711=1219.836,76.700,-46.678,-178.770,5.574,148.610
C08712=1219.831,76.949,-46.696,-178.768,5.574,148.609
C08713=1219.826,77.199,-46.714,-178.766,5.575,148.609
C08714=1219.822,77.448,-46.731,-178.763,5.576,148.608
C08715=1219.817,77.697,-46.749,-178.760,5.576,148.607
C08716=1219.812,77.947,-46.766,-178.758,5.577,148.607
C08717=1219.807,78.196,-46.784,-178.756,5.578,148.606
C08718=1219.802,78.445,-46.802,-178.752,5.579,148.605
C08719=1219.798,78.695,-46.821,-178.750,5.580,148.605
C08720=1219.793,78.944,-46.837,-178.748,5.581,148.604
C08721=1219.788,79.193,-46.855,-178.745,5.582,148.604
C08722=1219.783,79.443,-46.873,-178.742,5.582,148.603
C08723=1219.778,79.692,-46.891,-178.740,5.583,148.602
C08724=1219.773,79.942,-46.908,-178.738,5.584,148.602
C08725=1219.768,80.191,-46.926,-178.735,5.584,148.601
C08726=1219.763,80.440,-46.944,-178.732,5.586,148.601
C08727=1219.758,80.689,-46.962,-178.729,5.586,148.600
C08728=1219.753,80.939,-46.980,-178.727,5.587,148.600
C08729=1219.748,81.207,-46.999,-178.725,5.588,148.599
C08730=1219.743,81.475,-47.019,-178.722,5.588,148.598
C08731=1219.738,81.744,-47.038,-178.719,5.590,148.598
C08732=1219.733,82.013,-47.057,-178.716,5.590,148.597
C08733=1219.728,82.262,-47.075,-178.713,5.591,148.596
C08734=1219.723,82.511,-47.093,-178.711,5.592,148.596
C08735=1219.718,82.760,-47.111,-178.709,5.592,148.595
C08736=1219.714,83.009,-47.128,-178.705,5.594,148.595
C08737=1219.709,83.258,-47.146,-178.703,5.595,148.594
C08738=1219.704,83.508,-47.163,-178.701,5.595,148.594
C08739=1219.699,83.757,-47.181,-178.698,5.596,148.593
C08740=1219.694,84.006,-47.199,-178.695,5.597,148.592
C08741=1219.689,84.255,-47.217,-178.693,5.597,148.592
C08742=1219.685,84.505,-47.235,-178.691,5.598,148.591
C08743=1219.680,84.754,-47.253,-178.688,5.599,148.590
C08744=1219.675,85.004,-47.271,-178.685,5.600,148.590
C08745=1219.670,85.253,-47.289,-178.683,5.601,148.589
C08746=1219.665,85.502,-47.307,-178.680,5.602,148.589
C08747=1219.660,85.751,-47.325,-178.678,5.602,148.588
C08748=1219.654,86.001,-47.344,-178.675,5.603,148.588
C08749=1219.650,86.251,-47.362,-178.672,5.605,148.587
C08750=1219.645,86.500,-47.380,-178.670,5.605,148.586
C08751=1219.640,86.749,-47.398,-178.667,5.606,148.586
C08752=1219.635,86.998,-47.416,-178.665,5.607,148.585
C08753=1219.630,87.247,-47.434,-178.662,5.607,148.585
C08754=1219.625,87.496,-47.452,-178.660,5.608,148.584
C08755=1219.621,87.746,-47.470,-178.657,5.610,148.584
C08756=1219.616,87.995,-47.489,-178.654,5.610,148.583
C08757=1219.611,88.245,-47.506,-178.652,5.611,148.583
C08758=1219.606,88.494,-47.524,-178.650,5.612,148.582
C08759=1219.602,88.743,-47.542,-178.647,5.612,148.581
C08760=1219.597,88.992,-47.560,-178.645,5.613,148.581
C08761=1219.592,89.242,-47.579,-178.642,5.615,148.580
C08762=1219.587,89.492,-47.597,-178.639,5.615,148.579
C08763=1219.582,89.741,-47.615,-178.637,5.616,148.579
C08764=1219.577,89.989,-47.634,-178.634,5.617,148.578
C08765=1219.572,90.238,-47.652,-178.632,5.617,148.578
C08766=1219.568,90.488,-47.670,-178.628,5.619,148.577
C08767=1219.563,90.738,-47.688,-178.626,5.620,148.577
C08768=1219.558,90.987,-47.706,-178.624,5.620,148.576
C08769=1219.552,91.236,-47.725,-178.621,5.621,148.575
C08770=1219.548,91.485,-47.744,-178.619,5.622,148.575
C08771=1219.544,91.735,-47.762,-178.616,5.622,148.574
C08772=1219.539,91.984,-47.780,-178.613,5.624,148.574
C08773=1219.534,92.233,-47.798,-178.611,5.625,148.573
C08774=1219.528,92.482,-47.816,-178.608,5.625,148.573
C08775=1219.524,92.732,-47.836,-178.606,5.626,148.572
C08776=1219.519,92.981,-47.854,-178.604,5.627,148.572
C08777=1219.514,93.230,-47.871,-178.600,5.628,148.571
C08778=1219.509,93.479,-47.889,-178.598,5.629,148.570
C08779=1219.504,93.729,-47.908,-178.596,5.630,148.570
C08780=1219.500,93.978,-47.927,-178.593,5.630,148.569
C08781=1219.495,94.227,-47.945,-178.591,5.631,148.569
C08782=1219.490,94.477,-47.963,-178.588,5.633,148.568
C08783=1219.485,94.726,-47.983,-178.585,5.633,148.567
C08784=1219.480,94.975,-48.001,-178.583,5.634,148.567
C08785=1219.475,95.224,-48.019,-178.580,5.635,148.566
C08786=1219.471,95.474,-48.037,-178.578,5.636,148.566
C08787=1219.466,95.723,-48.056,-178.575,5.637,148.565
C08788=1219.461,95.972,-48.074,-178.572,5.638,148.565
C08789=1219.456,96.222,-48.093,-178.570,5.639,148.564
C08790=1219.451,96.471,-48.112,-178.568,5.639,148.564
C08791=1219.446,96.720,-48.130,-178.564,5.641,148.563
C08792=1219.442,96.969,-48.149,-178.562,5.642,148.562
C08793=1219.437,97.219,-48.167,-178.560,5.642,148.562
C08794=1219.432,97.468,-48.186,-178.557,5.643,148.561
C08795=1219.428,97.717,-48.205,-178.554,5.644,148.561
C08796=1219.423,97.966,-48.223,-178.552,5.645,148.560
C08797=1219.417,98.215,-48.242,-178.549,5.646,148.560
C08798=1219.413,98.465,-48.260,-178.547,5.647,148.559
C08799=1219.407,98.715,-48.279,-178.544,5.648,148.558
C08800=1219.403,98.963,-48.297,-178.541,5.649,148.558
C08801=1219.398,99.213,-48.316,-178.539,5.650,148.557
C08802=1219.393,99.462,-48.335,-178.536,5.651,148.557
C08803=1219.388,99.711,-48.353,-178.534,5.651,148.556
C08804=1219.384,99.960,-48.372,-178.532,5.652,148.556
C08805=1219.378,100.210,-48.391,-178.529,5.654,148.555
C08806=1219.374,100.458,-48.409,-178.526,5.654,148.554
C08807=1219.369,100.709,-48.428,-178.524,5.655,148.554
C08808=1219.364,100.957,-48.447,-178.521,5.656,148.553
C08809=1219.360,101.207,-48.465,-178.519,5.657,148.553
C08810=1219.355,101.456,-48.485,-178.516,5.658,148.552
C08811=1219.350,101.705,-48.503,-178.513,5.659,148.552
C08812=1219.345,101.955,-48.522,-178.511,5.660,148.551
C08813=1219.340,102.204,-48.540,-178.508,5.661,148.551
C08814=1219.335,102.453,-48.560,-178.506,5.662,148.550
C08815=1219.331,102.702,-48.579,-178.503,5.663,148.550
C08816=1219.326,102.951,-48.597,-178.501,5.663,148.549
C08817=1219.321,103.201,-48.616,-178.498,5.665,148.549
C08818=1219.316,103.450,-48.634,-178.495,5.666,148.548
C08819=1219.311,103.699,-48.654,-178.493,5.666,148.547
C08820=1219.307,103.948,-48.673,-178.491,5.667,148.547
C08821=1219.302,104.198,-48.692,-178.487,5.669,148.546
C08822=1219.297,104.447,-48.710,-178.485,5.669,148.546
C08823=1219.292,104.696,-48.730,-178.483,5.670,148.545
C08824=1219.287,104.946,-48.748,-178.479,5.672,148.544
C08825=1219.282,105.194,-48.767,-178.477,5.672,148.544
C08826=1219.278,105.444,-48.786,-178.475,5.673,148.543
C08827=1219.272,105.693,-48.805,-178.473,5.674,148.543
C08828=1219.268,105.942,-48.824,-178.469,5.675,148.542
C08829=1219.263,106.191,-48.843,-178.467,5.676,148.542
C08830=1219.258,106.441,-48.862,-178.465,5.677,148.541
C08831=1219.253,106.690,-48.881,-178.462,5.678,148.541
C08832=1219.249,106.940,-48.900,-178.459,5.679,148.540
C08833=1219.244,107.208,-48.920,-178.457,5.680,148.540
C08834=1219.239,107.476,-48.941,-178.454,5.681,148.539
C08835=1219.233,107.744,-48.962,-178.451,5.682,148.538
C08836=1219.227,108.013,-48.982,-178.448,5.683,148.538
C08837=1219.223,108.262,-49.001,-178.446,5.684,148.537
C08838=1219.218,108.511,-49.020,-178.443,5.685,148.537
C08839=1219.213,108.761,-49.040,-178.441,5.686,148.536
C08840=1219.209,109.010,-49.059,-178.438,5.687,148.536
C08841=1219.204,109.259,-49.077,-178.436,5.688,148.535
C08842=1219.200,109.509,-49.096,-178.433,5.689,148.535
C08843=1219.194,109.758,-49.116,-178.430,5.690,148.534
C08844=1219.190,110.007,-49.135,-178.428,5.691,148.534
C08845=1219.185,110.256,-49.154,-178.425,5.692,148.533
C08846=1219.180,110.505,-49.174,-178.423,5.693,148.532
C08847=1219.175,110.754,-49.193,-178.420,5.694,148.532
C08848=1219.171,111.004,-49.211,-178.417,5.695,148.531
C08849=1219.165,111.253,-49.231,-178.415,5.696,148.531
C08850=1219.160,111.502,-49.250,-178.412,5.697,148.530
C08851=1219.156,111.751,-49.269,-178.410,5.698,148.530
C08852=1219.151,112.001,-49.289,-178.407,5.699,148.529
C08853=1219.146,112.250,-49.308,-178.405,5.700,148.529
C08854=1219.142,112.499,-49.327,-178.402,5.701,148.528
C08855=1219.137,112.748,-49.347,-178.400,5.702,148.528
C08856=1219.132,112.997,-49.366,-178.397,5.703,148.527
C08857=1219.127,113.247,-49.386,-178.394,5.704,148.526
C08858=1219.122,113.495,-49.404,-178.392,5.705,148.526
C08859=1219.118,113.745,-49.424,-178.389,5.706,148.525
C08860=1219.113,113.994,-49.444,-178.386,5.708,148.525
C08861=1219.107,114.243,-49.463,-178.384,5.708,148.524
C08862=1219.103,114.492,-49.482,-178.382,5.709,148.524
C08863=1219.098,114.741,-49.501,-178.379,5.711,148.523
C08864=1219.093,114.991,-49.521,-178.376,5.711,148.523
C08865=1219.089,115.240,-49.541,-178.374,5.712,148.522
C08866=1219.084,115.489,-49.559,-178.371,5.714,148.522
C08867=1219.079,115.739,-49.579,-178.369,5.715,148.521
C08868=1219.074,115.987,-49.598,-178.366,5.715,148.521
C08869=1219.069,116.237,-49.618,-178.363,5.717,148.520
C08870=1219.064,116.487,-49.637,-178.361,5.718,148.519
C08871=1219.060,116.735,-49.656,-178.359,5.719,148.519
C08872=1219.055,116.984,-49.677,-178.355,5.720,148.518
C08873=1219.051,117.234,-49.696,-178.353,5.721,148.518
C08874=1219.045,117.483,-49.716,-178.351,5.722,148.517
C08875=1219.041,117.732,-49.735,-178.348,5.723,148.517
C08876=1219.036,117.982,-49.755,-178.345,5.724,148.516
C08877=1219.031,118.230,-49.774,-178.343,5.725,148.516
C08878=1219.026,118.480,-49.793,-178.340,5.726,148.515
C08879=1219.022,118.729,-49.814,-178.337,5.727,148.515
C08880=1219.017,118.978,-49.833,-178.335,5.728,148.514
C08881=1219.012,119.227,-49.852,-178.332,5.729,148.514
C08882=1219.007,119.477,-49.872,-178.330,5.730,148.513
C08883=1219.002,119.726,-49.891,-178.327,5.731,148.513
C08884=1218.997,119.975,-49.912,-178.325,5.733,148.512
C08885=1218.993,120.224,-49.931,-178.322,5.733,148.512
C08886=1218.988,120.473,-49.950,-178.320,5.734,148.511
C08887=1218.983,120.722,-49.970,-178.317,5.736,148.511
C08888=1218.979,120.971,-49.990,-178.315,5.737,148.510
C08889=1218.974,121.221,-50.010,-178.312,5.737,148.509
C08890=1218.969,121.470,-50.029,-178.309,5.739,148.509
C08891=1218.964,121.719,-50.049,-178.307,5.740,148.508
C08892=1218.960,121.968,-50.069,-178.304,5.742,148.508
C08893=1218.954,122.217,-50.088,-178.302,5.742,148.507
C08894=1218.950,122.467,-50.108,-178.299,5.743,148.507
C08895=1218.945,122.716,-50.128,-178.296,5.745,148.506
C08896=1218.940,122.965,-50.148,-178.294,5.746,148.506
C08897=1218.935,123.214,-50.167,-178.291,5.746,148.505
C08898=1218.931,123.463,-50.188,-178.288,5.748,148.505
C08899=1218.926,123.713,-50.207,-178.286,5.749,148.504
C08900=1218.921,123.962,-50.227,-178.284,5.749,148.504
C08901=1218.916,124.210,-50.247,-178.281,5.751,148.503
C08902=1218.911,124.460,-50.267,-178.278,5.752,148.503
C08903=1218.907,124.709,-50.287,-178.276,5.753,148.502
C08904=1218.902,124.958,-50.307,-178.273,5.754,148.502
C08905=1218.897,125.208,-50.326,-178.271,5.755,148.501
C08906=1218.892,125.456,-50.346,-178.268,5.756,148.501
C08907=1218.888,125.706,-50.366,-178.266,5.757,148.500
C08908=1218.883,125.955,-50.386,-178.262,5.759,148.500
C08909=1218.878,126.204,-50.406,-178.260,5.760,148.499
C08910=1218.874,126.453,-50.427,-178.258,5.761,148.499
C08911=1218.869,126.702,-50.446,-178.255,5.762,148.498
C08912=1218.864,126.951,-50.466,-178.253,5.763,148.498
C08913=1218.859,127.201,-50.486,-178.250,5.764,148.497
C08914=1218.855,127.450,-50.506,-178.248,5.766,148.497
C08915=1218.850,127.699,-50.526,-178.245,5.766,148.496
C08916=1218.845,127.948,-50.546,-178.242,5.768,148.496
C08917=1218.840,128.197,-50.566,-178.240,5.769,148.495
C08918=1218.835,128.446,-50.587,-178.238,5.770,148.495
C08919=1218.831,128.696,-50.606,-178.234,5.771,148.494
C08920=1218.826,128.945,-50.627,-178.232,5.772,148.494
C08921=1218.822,129.194,-50.647,-178.229,5.774,148.493
C08922=1218.816,129.443,-50.666,-178.227,5.774,148.493
C08923=1218.811,129.692,-50.687,-178.224,5.775,148.492
C08924=1218.806,129.941,-50.707,-178.222,5.777,148.492
C08925=1218.802,130.190,-50.727,-178.219,5.778,148.491
C08926=1218.798,130.439,-50.748,-178.217,5.779,148.491
C08927=1218.793,130.689,-50.767,-178.214,5.780,148.490
C08928=1218.788,130.938,-50.788,-178.211,5.782,148.490
C08929=1218.783,131.188,-50.808,-178.209,5.782,148.489
C08930=1218.778,131.436,-50.828,-178.207,5.783,148.489
C08931=1218.773,131.685,-50.848,-178.204,5.785,148.488
C08932=1218.769,131.934,-50.868,-178.201,5.786,148.488
C08933=1218.764,132.183,-50.888,-178.199,5.788,148.487
C08934=1218.759,132.433,-50.909,-178.196,5.788,148.486
C08935=1218.755,132.682,-50.930,-178.194,5.789,148.486
C08936=1218.750,132.931,-50.949,-178.191,5.791,148.485
C08937=1218.745,133.200,-50.972,-178.188,5.792,148.485
C08938=1218.740,133.468,-50.993,-178.185,5.793,148.484
C08939=1218.734,133.737,-51.015,-178.182,5.794,148.484
C08940=1218.729,134.005,-51.037,-178.180,5.795,148.483
C08941=1218.724,134.254,-51.057,-178.177,5.797,148.483
C08942=1218.720,134.503,-51.078,-178.175,5.798,148.482
C08943=1218.715,134.753,-51.099,-178.172,5.799,148.482
C08944=1218.710,135.002,-51.118,-178.170,5.800,148.481
C08945=1218.705,135.251,-51.139,-178.166,5.802,148.481
C08946=1218.701,135.500,-51.159,-178.164,5.803,148.480
C08947=1218.696,135.749,-51.180,-178.162,5.804,148.480
C08948=1218.691,135.998,-51.200,-178.159,5.805,148.479
C08949=1218.687,136.247,-51.221,-178.157,5.806,148.479
C08950=1218.681,136.497,-51.241,-178.154,5.808,148.478
C08951=1218.677,136.746,-51.261,-178.152,5.809,148.478
C08952=1218.673,136.995,-51.282,-178.148,5.810,148.477
C08953=1218.667,137.244,-51.303,-178.146,5.811,148.477
C08954=1218.663,137.493,-51.323,-178.144,5.813,148.477
C08955=1218.659,137.742,-51.343,-178.141,5.813,148.476
C08956=1218.653,137.991,-51.364,-178.138,5.815,148.476
C08957=1218.649,138.240,-51.385,-178.136,5.816,148.475
C08958=1218.644,138.490,-51.406,-178.134,5.817,148.475
C08959=1218.639,138.739,-51.426,-178.130,5.818,148.474
C08960=1218.635,138.988,-51.446,-178.128,5.819,148.474
C08961=1218.629,139.237,-51.467,-178.126,5.821,148.473
C08962=1218.625,139.486,-51.487,-178.123,5.822,148.473
C08963=1218.620,139.736,-51.508,-178.120,5.823,148.472
C08964=1218.615,139.985,-51.528,-178.118,5.824,148.472
C08965=1218.611,140.234,-51.549,-178.115,5.826,148.471
C08966=1218.606,140.483,-51.570,-178.113,5.827,148.470
C08967=1218.601,140.732,-51.590,-178.110,5.828,148.470
C08968=1218.596,140.981,-51.611,-178.108,5.829,148.470
C08969=1218.592,141.229,-51.632,-178.105,5.831,148.469
C08970=1218.587,141.479,-51.653,-178.103,5.832,148.469
C08971=1218.582,141.728,-51.673,-178.099,5.833,148.468
C08972=1218.577,141.977,-51.694,-178.097,5.834,148.468
C08973=1218.573,142.226,-51.715,-178.095,5.836,148.467
C08974=1218.568,142.475,-51.736,-178.092,5.837,148.467
C08975=1218.563,142.724,-51.756,-178.089,5.838,148.466
C08976=1218.559,142.974,-51.777,-178.087,5.839,148.466
C08977=1218.554,143.223,-51.798,-178.084,5.841,148.465
C08978=1218.549,143.472,-51.819,-178.082,5.842,148.465
C08979=1218.545,143.721,-51.839,-178.079,5.843,148.464
C08980=1218.540,143.970,-51.861,-178.077,5.844,148.464
C08981=1218.535,144.219,-51.881,-178.074,5.845,148.463
C08982=1218.530,144.468,-51.902,-178.071,5.847,148.463
C08983=1218.526,144.717,-51.923,-178.069,5.848,148.463
C08984=1218.520,144.966,-51.944,-178.066,5.849,148.462
C08985=1218.516,145.215,-51.964,-178.064,5.850,148.461
C08986=1218.512,145.464,-51.986,-178.061,5.852,148.461
C08987=1218.507,145.713,-52.006,-178.059,5.853,148.460
C08988=1218.502,145.963,-52.027,-178.056,5.854,148.460
C08989=1218.497,146.212,-52.048,-178.053,5.856,148.460
C08990=1218.493,146.460,-52.069,-178.051,5.857,148.459
C08991=1218.488,146.709,-52.090,-178.048,5.859,148.459
C08992=1218.483,146.958,-52.111,-178.046,5.859,148.458
C08993=1218.479,147.208,-52.132,-178.043,5.861,148.458
C08994=1218.474,147.457,-52.154,-178.041,5.862,148.457
C08995=1218.469,147.706,-52.174,-178.038,5.863,148.457
C08996=1218.464,147.955,-52.195,-178.035,5.864,148.456
C08997=1218.460,148.204,-52.216,-178.032,5.866,148.456
C08998=1218.455,148.453,-52.237,-178.030,5.867,148.455
C08999=1218.450,148.703,-52.258,-178.028,5.869,148.455
C09000=1218.446,148.951,-52.280,-178.025,5.869,148.454
C09001=1218.441,149.200,-52.300,-178.022,5.871,148.454
C09002=1218.436,149.450,-52.321,-178.020,5.872,148.454
C09003=1218.432,149.698,-52.343,-178.017,5.874,148.453
C09004=1218.426,149.947,-52.363,-178.015,5.875,148.453
C09005=1218.422,150.197,-52.385,-178.012,5.876,148.452
C09006=1218.417,150.446,-52.407,-178.010,5.877,148.452
C09007=1218.413,150.695,-52.427,-178.007,5.879,148.451
C09008=1218.408,150.943,-52.449,-178.005,5.880,148.451
C09009=1218.403,151.193,-52.470,-178.002,5.881,148.450
C09010=1218.399,151.442,-52.491,-177.999,5.883,148.450
C09011=1218.394,151.691,-52.512,-177.996,5.884,148.449
C09012=1218.389,151.940,-52.533,-177.994,5.886,148.449
C09013=1218.384,152.189,-52.555,-177.992,5.887,148.448
C09014=1218.380,152.439,-52.575,-177.989,5.888,148.448
C09015=1218.375,152.687,-52.597,-177.986,5.889,148.447
C09016=1218.370,152.936,-52.618,-177.984,5.891,148.447
C09017=1218.365,153.185,-52.640,-177.981,5.891,148.446
C09018=1218.360,153.435,-52.661,-177.978,5.893,148.446
C09019=1218.356,153.683,-52.682,-177.976,5.894,148.446
C09020=1218.351,153.932,-52.704,-177.973,5.896,148.445
C09021=1218.346,154.181,-52.725,-177.971,5.898,148.445
C09022=1218.342,154.431,-52.747,-177.968,5.898,148.444
C09023=1218.337,154.680,-52.768,-177.965,5.900,148.444
C09024=1218.333,154.928,-52.789,-177.963,5.901,148.443
C09025=1218.328,155.177,-52.810,-177.961,5.903,148.443
C09026=1218.323,155.427,-52.832,-177.958,5.903,148.442
C09027=1218.318,155.675,-52.854,-177.955,5.905,148.442
C09028=1218.313,155.925,-52.875,-177.953,5.907,148.442
C09029=1218.309,156.174,-52.897,-177.950,5.908,148.441
C09030=1218.305,156.423,-52.917,-177.947,5.909,148.441
C09031=1218.300,156.672,-52.939,-177.945,5.910,148.440
C09032=1218.295,156.921,-52.961,-177.943,5.912,148.440
C09033=1218.290,157.170,-52.982,-177.940,5.913,148.439
C09034=1218.285,157.419,-53.003,-177.937,5.915,148.439
C09035=1218.281,157.668,-53.025,-177.935,5.917,148.438
C09036=1218.276,157.917,-53.047,-177.932,5.917,148.438
C09037=1218.271,158.166,-53.068,-177.929,5.919,148.437
C09038=1218.267,158.415,-53.090,-177.927,5.920,148.437
C09039=1218.262,158.664,-53.112,-177.924,5.921,148.437
C09040=1218.257,158.913,-53.132,-177.922,5.922,148.436
C09041=1218.252,159.182,-53.156,-177.919,5.924,148.436
C09042=1218.247,159.451,-53.180,-177.916,5.926,148.435
C09043=1218.242,159.720,-53.202,-177.914,5.928,148.435
C09044=1218.237,159.989,-53.226,-177.910,5.929,148.434
C09045=1218.233,160.238,-53.248,-177.908,5.930,148.434
C09046=1218.227,160.488,-53.269,-177.906,5.932,148.433
C09047=1218.223,160.736,-53.291,-177.903,5.932,148.433
C09048=1218.218,160.986,-53.313,-177.900,5.934,148.432
C09049=1218.213,161.234,-53.335,-177.898,5.936,148.432
C09050=1218.209,161.483,-53.357,-177.895,5.937,148.431
C09051=1218.204,161.733,-53.378,-177.892,5.939,148.431
C09052=1218.199,161.981,-53.399,-177.890,5.940,148.431
C09053=1218.195,162.231,-53.422,-177.888,5.941,148.430
C09054=1218.190,162.479,-53.443,-177.885,5.943,148.430
C09055=1218.186,162.729,-53.465,-177.882,5.944,148.429
C09056=1218.181,162.977,-53.487,-177.880,5.946,148.429
C09057=1218.176,163.226,-53.509,-177.877,5.947,148.428
C09058=1218.172,163.475,-53.531,-177.875,5.948,148.428
C09059=1218.167,163.724,-53.552,-177.872,5.950,148.428
C09060=1218.163,163.973,-53.574,-177.870,5.951,148.427
C09061=1218.158,164.222,-53.596,-177.867,5.952,148.427
C09062=1218.153,164.471,-53.618,-177.864,5.954,148.426
C09063=1218.149,164.720,-53.640,-177.862,5.955,148.426
C09064=1218.144,164.969,-53.662,-177.859,5.957,148.426
C09065=1218.139,165.218,-53.684,-177.856,5.958,148.425
C09066=1218.134,165.467,-53.706,-177.854,5.959,148.425
C09067=1218.130,165.716,-53.728,-177.851,5.961,148.424
C09068=1218.125,165.965,-53.750,-177.849,5.962,148.424
C09069=1218.120,166.214,-53.772,-177.846,5.964,148.423
C09070=1218.116,166.463,-53.793,-177.843,5.966,148.423
C09071=1218.111,166.712,-53.815,-177.841,5.967,148.422
C09072=1218.106,166.961,-53.837,-177.838,5.968,148.422
C09073=1218.101,167.210,-53.860,-177.835,5.970,148.422
C09074=1218.097,167.459,-53.881,-177.833,5.971,148.421
C09075=1218.092,167.708,-53.903,-177.831,5.973,148.421
C09076=1218.087,167.957,-53.925,-177.828,5.974,148.420
C09077=1218.083,168.206,-53.947,-177.825,5.975,148.420
C09078=1218.078,168.455,-53.969,-177.823,5.977,148.419
C09079=1218.074,168.704,-53.992,-177.820,5.979,148.419
C09080=1218.069,168.953,-54.014,-177.818,5.980,148.419
C09081=1218.064,169.202,-54.036,-177.815,5.981,148.418
C09082=1218.060,169.451,-54.058,-177.813,5.982,148.418
C09083=1218.055,169.700,-54.080,-177.810,5.984,148.417
C09084=1218.050,169.949,-54.102,-177.807,5.986,148.417
C09085=1218.046,170.198,-54.125,-177.805,5.987,148.416
C09086=1218.041,170.447,-54.147,-177.802,5.988,148.416
C09087=1218.036,170.696,-54.169,-177.800,5.990,148.416
C09088=1218.032,170.945,-54.191,-177.797,5.991,148.415
C09089=1218.027,171.194,-54.213,-177.794,5.993,148.415
C09090=1218.023,171.443,-54.236,-177.792,5.994,148.414
C09091=1218.017,171.692,-54.258,-177.790,5.995,148.414
C09092=1218.013,171.941,-54.280,-177.787,5.997,148.414
C09093=1218.008,172.190,-54.302,-177.784,5.999,148.413
C09094=1218.003,172.439,-54.325,-177.782,6.000,148.413
C09095=1217.999,172.688,-54.347,-177.779,6.002,148.412
C09096=1217.994,172.937,-54.369,-177.776,6.003,148.412
C09097=1217.990,173.185,-54.391,-177.774,6.004,148.411
C09098=1217.985,173.434,-54.414,-177.771,6.006,148.411
C09099=1217.980,173.684,-54.436,-177.768,6.008,148.411
C09100=1217.976,173.933,-54.459,-177.766,6.010,148.410
C09101=1217.971,174.181,-54.481,-177.764,6.011,148.410
C09102=1217.966,174.431,-54.503,-177.761,6.012,148.409
C09103=1217.961,174.679,-54.526,-177.758,6.014,148.409
C09104=1217.957,174.928,-54.548,-177.756,6.015,148.408
C09105=1217.953,175.177,-54.571,-177.753,6.017,148.408
C09106=1217.947,175.426,-54.593,-177.751,6.018,148.408
C09107=1217.943,175.675,-54.615,-177.748,6.019,148.407
C09108=1217.938,175.924,-54.638,-177.745,6.021,148.407
C09109=1217.934,176.173,-54.660,-177.743,6.023,148.406
C09110=1217.930,176.422,-54.683,-177.741,6.024,148.406
C09111=1217.925,176.671,-54.705,-177.738,6.026,148.406
C09112=1217.920,176.919,-54.728,-177.735,6.027,148.405
C09113=1217.915,177.169,-54.750,-177.732,6.029,148.405
C09114=1217.911,177.418,-54.773,-177.730,6.030,148.404
C09115=1217.905,177.667,-54.795,-177.727,6.032,148.404
C09116=1217.901,177.915,-54.818,-177.725,6.034,148.404
C09117=1217.897,178.165,-54.840,-177.723,6.035,148.403
C09118=1217.892,178.413,-54.863,-177.720,6.036,148.403
C09119=1217.888,178.663,-54.885,-177.717,6.038,148.402
C09120=1217.883,178.912,-54.909,-177.714,6.040,148.402
C09121=1217.878,179.160,-54.930,-177.712,6.041,148.402
C09122=1217.873,179.409,-54.954,-177.709,6.043,148.401
C09123=1217.869,179.658,-54.976,-177.707,6.044,148.401
C09124=1217.864,179.908,-54.999,-177.704,6.045,148.400
C09125=1217.860,180.156,-55.022,-177.701,6.047,148.400
C09126=1217.855,180.405,-55.044,-177.699,6.049,148.400
C09127=1217.851,180.654,-55.067,-177.696,6.051,148.399
C09128=1217.846,180.902,-55.090,-177.694,6.052,148.399
C09129=1217.841,181.152,-55.112,-177.691,6.053,148.398
C09130=1217.837,181.401,-55.135,-177.688,6.055,148.398
C09131=1217.832,181.650,-55.159,-177.686,6.057,148.398
C09132=1217.827,181.898,-55.180,-177.684,6.058,148.397
